Yaskawa INFORM job: A_ROOF_UPPER_0614_2_PAINT_0.JBI

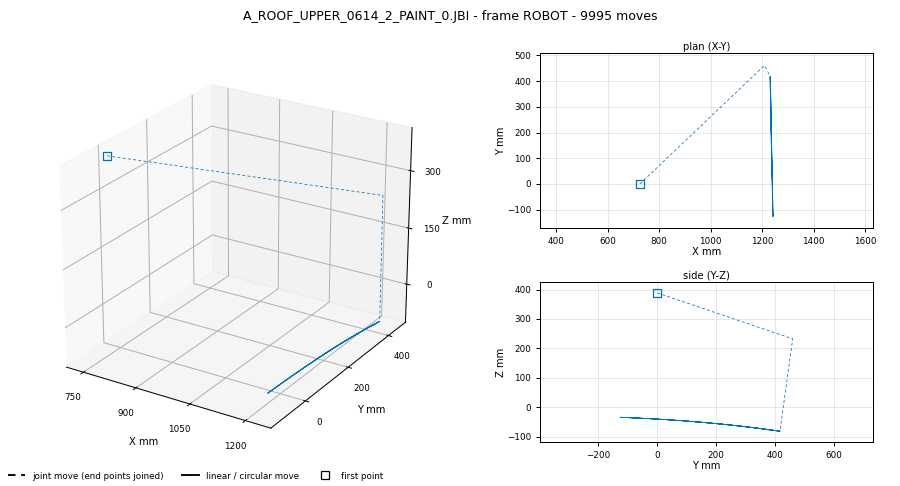
[picture p0: tool path of A_ROOF_UPPER_0614_2_PAINT_0.JBI in frame ROBOT, 9995 of 9995 moves have a stored position in this frame; points joined in program order, loops and branches not executed]
/JOB
//NAME A_ROOF_UPPER_0614_2_PAINT
//POS
///NPOS 9995,0,0,0,0,0
///TOOL 0
///USER 0
///POSTYPE ROBOT
///RECTAN
///RCONF 1,0,0,0,0,0,0,0,0,0,0,0,0,0,0,0,0,0,0,0,0,0,0,0
C00000=725.000,0.000,388.500,-180.000,-0.000,0.000
///TOOL 1
///USER 0
///POSTYPE ROBOT
///RECTAN
C00001=1208.850,460.483,232.516,-175.614,7.825,148.236
C00002=1232.740,417.098,-81.457,-175.614,7.825,148.236
C00003=1232.746,416.739,-81.407,-175.614,7.822,148.236
C00004=1232.752,416.380,-81.357,-175.615,7.819,148.235
C00005=1232.757,416.020,-81.307,-175.616,7.816,148.234
C00006=1232.764,415.662,-81.256,-175.617,7.813,148.234
C00007=1232.767,415.414,-81.222,-175.617,7.811,148.234
C00008=1232.771,415.166,-81.188,-175.619,7.808,148.233
C00009=1232.775,414.918,-81.153,-175.619,7.806,148.233
C00010=1232.779,414.671,-81.119,-175.619,7.804,148.232
C00011=1232.784,414.424,-81.085,-175.620,7.802,148.232
C00012=1232.788,414.176,-81.050,-175.621,7.800,148.232
C00013=1232.792,413.929,-81.016,-175.621,7.798,148.231
C00014=1232.796,413.680,-80.981,-175.621,7.796,148.231
C00015=1232.800,413.433,-80.947,-175.623,7.793,148.230
C00016=1232.804,413.186,-80.913,-175.623,7.791,148.230
C00017=1232.808,412.938,-80.878,-175.624,7.789,148.230
C00018=1232.813,412.690,-80.843,-175.625,7.787,148.229
C00019=1232.816,412.443,-80.809,-175.625,7.785,148.229
C00020=1232.820,412.195,-80.775,-175.626,7.782,148.228
C00021=1232.825,411.948,-80.740,-175.626,7.780,148.228
C00022=1232.828,411.700,-80.706,-175.627,7.778,148.228
C00023=1232.833,411.452,-80.672,-175.628,7.776,148.227
C00024=1232.836,411.205,-80.637,-175.628,7.774,148.227
C00025=1232.841,410.957,-80.603,-175.629,7.772,148.226
C00026=1232.845,410.710,-80.568,-175.630,7.769,148.226
C00027=1232.848,410.462,-80.534,-175.630,7.767,148.226
C00028=1232.853,410.214,-80.500,-175.631,7.765,148.225
C00029=1232.856,409.966,-80.466,-175.631,7.763,148.225
C00030=1232.861,409.719,-80.432,-175.632,7.760,148.224
C00031=1232.866,409.471,-80.397,-175.633,7.758,148.224
C00032=1232.869,409.224,-80.363,-175.634,7.756,148.224
C00033=1232.873,408.976,-80.329,-175.634,7.754,148.223
C00034=1232.877,408.729,-80.295,-175.634,7.752,148.223
C00035=1232.881,408.481,-80.260,-175.635,7.749,148.222
C00036=1232.886,408.233,-80.225,-175.636,7.747,148.222
C00037=1232.890,407.986,-80.191,-175.637,7.745,148.222
C00038=1232.894,407.738,-80.157,-175.637,7.743,148.221
C00039=1232.898,407.491,-80.123,-175.638,7.740,148.221
C00040=1232.902,407.243,-80.089,-175.639,7.738,148.220
C00041=1232.905,406.995,-80.055,-175.639,7.736,148.220
C00042=1232.910,406.748,-80.020,-175.640,7.734,148.220
C00043=1232.914,406.501,-79.986,-175.641,7.731,148.219
C00044=1232.918,406.253,-79.952,-175.641,7.729,148.219
C00045=1232.923,406.005,-79.918,-175.642,7.727,148.218
C00046=1232.927,405.757,-79.884,-175.643,7.724,148.218
C00047=1232.931,405.509,-79.849,-175.644,7.722,148.218
C00048=1232.934,405.262,-79.815,-175.644,7.720,148.217
C00049=1232.939,405.015,-79.781,-175.644,7.718,148.217
C00050=1232.942,404.766,-79.747,-175.646,7.715,148.216
C00051=1232.947,404.519,-79.713,-175.646,7.713,148.216
C00052=1232.951,404.272,-79.679,-175.647,7.711,148.216
C00053=1232.955,404.024,-79.644,-175.648,7.708,148.215
C00054=1232.959,403.777,-79.610,-175.649,7.706,148.215
C00055=1232.964,403.529,-79.576,-175.649,7.704,148.214
C00056=1232.967,403.281,-79.542,-175.650,7.701,148.214
C00057=1232.971,403.033,-79.508,-175.651,7.699,148.214
C00058=1232.975,402.786,-79.474,-175.651,7.697,148.213
C00059=1232.979,402.538,-79.440,-175.652,7.694,148.213
C00060=1232.983,402.290,-79.406,-175.653,7.692,148.212
C00061=1232.988,402.043,-79.371,-175.653,7.690,148.212
C00062=1232.991,401.795,-79.337,-175.654,7.687,148.212
C00063=1232.996,401.547,-79.303,-175.655,7.685,148.211
C00064=1233.000,401.300,-79.270,-175.656,7.683,148.211
C00065=1233.004,401.053,-79.236,-175.657,7.681,148.211
C00066=1233.008,400.804,-79.202,-175.657,7.678,148.210
C00067=1233.012,400.557,-79.168,-175.658,7.676,148.210
C00068=1233.016,400.310,-79.133,-175.659,7.673,148.209
C00069=1233.020,400.061,-79.100,-175.659,7.671,148.209
C00070=1233.024,399.814,-79.065,-175.660,7.669,148.209
C00071=1233.028,399.567,-79.031,-175.661,7.667,148.208
C00072=1233.033,399.319,-78.998,-175.662,7.665,148.208
C00073=1233.036,399.071,-78.963,-175.662,7.662,148.207
C00074=1233.040,398.824,-78.930,-175.663,7.660,148.207
C00075=1233.045,398.576,-78.896,-175.664,7.658,148.206
C00076=1233.049,398.329,-78.862,-175.665,7.655,148.206
C00077=1233.053,398.080,-78.827,-175.666,7.653,148.206
C00078=1233.057,397.833,-78.794,-175.667,7.650,148.205
C00079=1233.061,397.586,-78.760,-175.667,7.648,148.205
C00080=1233.066,397.338,-78.726,-175.668,7.645,148.204
C00081=1233.069,397.090,-78.692,-175.669,7.643,148.204
C00082=1233.074,396.842,-78.658,-175.669,7.641,148.204
C00083=1233.078,396.595,-78.624,-175.670,7.638,148.203
C00084=1233.081,396.348,-78.591,-175.671,7.636,148.203
C00085=1233.086,396.099,-78.556,-175.672,7.633,148.203
C00086=1233.090,395.852,-78.523,-175.673,7.631,148.202
C00087=1233.094,395.604,-78.489,-175.674,7.628,148.202
C00088=1233.098,395.357,-78.455,-175.674,7.626,148.201
C00089=1233.102,395.108,-78.421,-175.675,7.623,148.201
C00090=1233.106,394.861,-78.388,-175.676,7.621,148.201
C00091=1233.111,394.613,-78.354,-175.677,7.619,148.200
C00092=1233.114,394.366,-78.320,-175.678,7.617,148.200
C00093=1233.119,394.118,-78.286,-175.678,7.615,148.199
C00094=1233.122,393.870,-78.252,-175.680,7.612,148.199
C00095=1233.127,393.589,-78.213,-175.681,7.609,148.199
C00096=1233.132,393.307,-78.175,-175.681,7.606,148.198
C00097=1233.136,393.027,-78.137,-175.682,7.604,148.198
C00098=1233.141,392.746,-78.099,-175.683,7.601,148.197
C00099=1233.145,392.498,-78.065,-175.684,7.598,148.197
C00100=1233.150,392.250,-78.031,-175.685,7.596,148.197
C00101=1233.153,392.003,-77.997,-175.686,7.593,148.196
C00102=1233.158,391.755,-77.964,-175.687,7.591,148.196
C00103=1233.162,391.507,-77.931,-175.688,7.589,148.195
C00104=1233.166,391.259,-77.896,-175.689,7.586,148.195
C00105=1233.170,391.011,-77.863,-175.690,7.584,148.195
C00106=1233.174,390.764,-77.829,-175.691,7.581,148.194
C00107=1233.178,390.516,-77.795,-175.691,7.579,148.194
C00108=1233.183,390.268,-77.762,-175.692,7.576,148.193
C00109=1233.186,390.021,-77.728,-175.693,7.574,148.193
C00110=1233.190,389.773,-77.695,-175.694,7.571,148.193
C00111=1233.195,389.525,-77.660,-175.695,7.569,148.192
C00112=1233.199,389.278,-77.627,-175.696,7.566,148.192
C00113=1233.203,389.030,-77.594,-175.697,7.563,148.191
C00114=1233.207,388.783,-77.560,-175.697,7.561,148.191
C00115=1233.212,388.535,-77.526,-175.699,7.559,148.191
C00116=1233.215,388.286,-77.493,-175.699,7.557,148.190
C00117=1233.219,388.039,-77.459,-175.700,7.554,148.190
C00118=1233.223,387.792,-77.426,-175.702,7.551,148.189
C00119=1233.227,387.544,-77.393,-175.702,7.549,148.189
C00120=1233.232,387.296,-77.358,-175.703,7.546,148.189
C00121=1233.236,387.049,-77.325,-175.704,7.544,148.188
C00122=1233.240,386.801,-77.292,-175.705,7.541,148.188
C00123=1233.243,386.553,-77.258,-175.706,7.538,148.188
C00124=1233.247,386.305,-77.224,-175.707,7.536,148.187
C00125=1233.252,386.057,-77.191,-175.708,7.534,148.187
C00126=1233.256,385.810,-77.158,-175.710,7.531,148.187
C00127=1233.260,385.563,-77.124,-175.710,7.529,148.186
C00128=1233.264,385.315,-77.091,-175.711,7.526,148.186
C00129=1233.269,385.067,-77.057,-175.713,7.524,148.186
C00130=1233.273,384.819,-77.024,-175.713,7.522,148.185
C00131=1233.277,384.571,-76.989,-175.714,7.519,148.185
C00132=1233.281,384.324,-76.956,-175.715,7.517,148.184
C00133=1233.285,384.076,-76.923,-175.716,7.514,148.184
C00134=1233.289,383.828,-76.890,-175.717,7.511,148.184
C00135=1233.293,383.580,-76.857,-175.719,7.508,148.183
C00136=1233.297,383.333,-76.823,-175.719,7.506,148.183
C00137=1233.301,383.086,-76.790,-175.720,7.503,148.182
C00138=1233.306,382.837,-76.756,-175.721,7.501,148.182
C00139=1233.310,382.590,-76.723,-175.723,7.499,148.182
C00140=1233.314,382.341,-76.689,-175.724,7.496,148.182
C00141=1233.318,382.094,-76.656,-175.725,7.493,148.181
C00142=1233.322,381.846,-76.623,-175.725,7.491,148.181
C00143=1233.326,381.599,-76.589,-175.727,7.488,148.180
C00144=1233.330,381.351,-76.556,-175.728,7.486,148.180
C00145=1233.334,381.103,-76.523,-175.729,7.483,148.180
C00146=1233.338,380.856,-76.490,-175.730,7.481,148.179
C00147=1233.342,380.608,-76.457,-175.731,7.478,148.179
C00148=1233.347,380.360,-76.423,-175.732,7.475,148.179
C00149=1233.351,380.112,-76.390,-175.733,7.473,148.178
C00150=1233.356,379.864,-76.356,-175.734,7.471,148.178
C00151=1233.360,379.617,-76.323,-175.735,7.468,148.178
C00152=1233.364,379.369,-76.290,-175.736,7.465,148.177
C00153=1233.368,379.121,-76.257,-175.738,7.462,148.177
C00154=1233.372,378.874,-76.223,-175.739,7.460,148.177
C00155=1233.376,378.626,-76.190,-175.740,7.458,148.176
C00156=1233.379,378.378,-76.156,-175.741,7.455,148.176
C00157=1233.384,378.130,-76.123,-175.742,7.452,148.175
C00158=1233.388,377.882,-76.090,-175.743,7.450,148.175
C00159=1233.392,377.635,-76.057,-175.744,7.447,148.175
C00160=1233.396,377.387,-76.024,-175.746,7.445,148.174
C00161=1233.400,377.139,-75.991,-175.747,7.442,148.174
C00162=1233.404,376.891,-75.957,-175.748,7.439,148.174
C00163=1233.408,376.644,-75.924,-175.749,7.437,148.173
C00164=1233.413,376.395,-75.892,-175.750,7.434,148.173
C00165=1233.417,376.148,-75.859,-175.751,7.432,148.173
C00166=1233.421,375.900,-75.826,-175.753,7.429,148.173
C00167=1233.425,375.652,-75.792,-175.754,7.426,148.172
C00168=1233.429,375.404,-75.759,-175.755,7.423,148.172
C00169=1233.434,375.157,-75.726,-175.756,7.421,148.171
C00170=1233.438,374.909,-75.693,-175.757,7.419,148.171
C00171=1233.442,374.661,-75.660,-175.759,7.416,148.171
C00172=1233.446,374.414,-75.627,-175.760,7.413,148.170
C00173=1233.450,374.166,-75.594,-175.761,7.411,148.170
C00174=1233.454,373.918,-75.560,-175.763,7.408,148.170
C00175=1233.458,373.670,-75.528,-175.763,7.406,148.169
C00176=1233.462,373.422,-75.495,-175.765,7.403,148.169
C00177=1233.466,373.175,-75.462,-175.766,7.401,148.169
C00178=1233.470,372.927,-75.429,-175.767,7.398,148.168
C00179=1233.474,372.679,-75.396,-175.769,7.395,148.168
C00180=1233.479,372.431,-75.363,-175.770,7.392,148.168
C00181=1233.483,372.183,-75.330,-175.771,7.390,148.168
C00182=1233.487,371.935,-75.297,-175.773,7.387,148.167
C00183=1233.492,371.688,-75.264,-175.773,7.385,148.167
C00184=1233.496,371.441,-75.231,-175.775,7.383,148.167
C00185=1233.499,371.193,-75.199,-175.776,7.380,148.166
C00186=1233.504,370.945,-75.166,-175.777,7.377,148.166
C00187=1233.508,370.697,-75.133,-175.779,7.374,148.166
C00188=1233.512,370.449,-75.100,-175.780,7.371,148.165
C00189=1233.516,370.202,-75.067,-175.782,7.369,148.165
C00190=1233.521,369.953,-75.034,-175.783,7.366,148.165
C00191=1233.525,369.706,-75.001,-175.784,7.364,148.165
C00192=1233.528,369.458,-74.969,-175.785,7.361,148.164
C00193=1233.532,369.210,-74.935,-175.787,7.358,148.164
C00194=1233.537,368.962,-74.903,-175.788,7.355,148.164
C00195=1233.541,368.714,-74.870,-175.790,7.353,148.163
C00196=1233.545,368.467,-74.837,-175.790,7.351,148.163
C00197=1233.549,368.219,-74.805,-175.792,7.348,148.163
C00198=1233.554,367.972,-74.772,-175.793,7.346,148.162
C00199=1233.558,367.692,-74.734,-175.795,7.342,148.162
C00200=1233.563,367.412,-74.698,-175.797,7.339,148.162
C00201=1233.568,367.133,-74.661,-175.798,7.336,148.161
C00202=1233.572,366.854,-74.624,-175.800,7.333,148.161
C00203=1233.577,366.605,-74.591,-175.801,7.330,148.161
C00204=1233.580,366.358,-74.559,-175.803,7.328,148.161
C00205=1233.585,366.110,-74.526,-175.804,7.325,148.160
C00206=1233.589,365.862,-74.493,-175.805,7.322,148.160
C00207=1233.594,365.614,-74.461,-175.807,7.320,148.160
C00208=1233.597,365.367,-74.428,-175.808,7.317,148.159
C00209=1233.601,365.119,-74.395,-175.810,7.314,148.159
C00210=1233.606,364.871,-74.363,-175.811,7.312,148.159
C00211=1233.610,364.623,-74.330,-175.813,7.309,148.159
C00212=1233.614,364.376,-74.298,-175.814,7.307,148.158
C00213=1233.618,364.128,-74.265,-175.815,7.304,148.158
C00214=1233.623,363.879,-74.233,-175.817,7.301,148.158
C00215=1233.626,363.632,-74.200,-175.818,7.298,148.157
C00216=1233.631,363.384,-74.168,-175.820,7.296,148.157
C00217=1233.635,363.136,-74.134,-175.821,7.293,148.157
C00218=1233.639,362.889,-74.103,-175.823,7.291,148.157
C00219=1233.643,362.641,-74.070,-175.824,7.288,148.156
C00220=1233.648,362.393,-74.037,-175.826,7.285,148.156
C00221=1233.651,362.145,-74.005,-175.827,7.283,148.156
C00222=1233.655,361.897,-73.972,-175.829,7.280,148.156
C00223=1233.660,361.648,-73.940,-175.830,7.278,148.156
C00224=1233.664,361.402,-73.908,-175.831,7.275,148.155
C00225=1233.668,361.153,-73.875,-175.833,7.272,148.155
C00226=1233.672,360.906,-73.842,-175.835,7.270,148.155
C00227=1233.676,360.658,-73.810,-175.836,7.267,148.155
C00228=1233.681,360.409,-73.778,-175.837,7.264,148.154
C00229=1233.685,360.162,-73.745,-175.839,7.262,148.154
C00230=1233.689,359.914,-73.713,-175.841,7.259,148.154
C00231=1233.693,359.666,-73.681,-175.842,7.257,148.154
C00232=1233.697,359.418,-73.648,-175.843,7.254,148.153
C00233=1233.702,359.171,-73.616,-175.846,7.250,148.153
C00234=1233.706,358.922,-73.584,-175.847,7.248,148.153
C00235=1233.710,358.675,-73.551,-175.849,7.245,148.153
C00236=1233.714,358.427,-73.519,-175.850,7.243,148.152
C00237=1233.718,358.179,-73.487,-175.852,7.240,148.152
C00238=1233.723,357.932,-73.454,-175.853,7.238,148.152
C00239=1233.727,357.683,-73.422,-175.855,7.235,148.152
C00240=1233.731,357.435,-73.390,-175.856,7.232,148.151
C00241=1233.735,357.187,-73.357,-175.858,7.230,148.151
C00242=1233.739,356.940,-73.325,-175.859,7.227,148.151
C00243=1233.744,356.692,-73.293,-175.861,7.225,148.151
C00244=1233.747,356.444,-73.261,-175.862,7.222,148.150
C00245=1233.752,356.195,-73.228,-175.865,7.219,148.150
C00246=1233.756,355.949,-73.196,-175.866,7.216,148.150
C00247=1233.760,355.700,-73.164,-175.868,7.214,148.150
C00248=1233.764,355.452,-73.132,-175.869,7.211,148.150
C00249=1233.769,355.205,-73.100,-175.871,7.208,148.149
C00250=1233.773,354.957,-73.068,-175.872,7.206,148.149
C00251=1233.777,354.708,-73.035,-175.874,7.203,148.149
C00252=1233.781,354.461,-73.003,-175.875,7.201,148.149
C00253=1233.786,354.213,-72.971,-175.877,7.198,148.149
C00254=1233.789,353.965,-72.939,-175.879,7.196,148.148
C00255=1233.794,353.717,-72.907,-175.881,7.192,148.148
C00256=1233.798,353.469,-72.875,-175.882,7.190,148.148
C00257=1233.802,353.221,-72.843,-175.884,7.187,148.148
C00258=1233.806,352.973,-72.811,-175.886,7.185,148.148
C00259=1233.810,352.725,-72.779,-175.887,7.182,148.147
C00260=1233.815,352.477,-72.747,-175.889,7.180,148.147
C00261=1233.819,352.229,-72.715,-175.891,7.177,148.147
C00262=1233.823,351.981,-72.683,-175.892,7.174,148.147
C00263=1233.827,351.734,-72.650,-175.894,7.171,148.147
C00264=1233.831,351.486,-72.619,-175.896,7.169,148.146
C00265=1233.835,351.238,-72.586,-175.898,7.166,148.146
C00266=1233.840,350.991,-72.555,-175.899,7.163,148.146
C00267=1233.843,350.743,-72.523,-175.901,7.161,148.146
C00268=1233.848,350.494,-72.490,-175.902,7.158,148.146
C00269=1233.852,350.247,-72.459,-175.904,7.156,148.145
C00270=1233.856,349.999,-72.427,-175.906,7.152,148.145
C00271=1233.861,349.750,-72.395,-175.908,7.150,148.145
C00272=1233.865,349.502,-72.364,-175.909,7.147,148.145
C00273=1233.869,349.254,-72.332,-175.911,7.145,148.145
C00274=1233.874,349.007,-72.300,-175.913,7.142,148.145
C00275=1233.877,348.759,-72.268,-175.914,7.140,148.144
C00276=1233.881,348.511,-72.236,-175.916,7.137,148.144
C00277=1233.886,348.263,-72.204,-175.918,7.134,148.144
C00278=1233.890,348.015,-72.172,-175.920,7.131,148.144
C00279=1233.893,347.767,-72.140,-175.921,7.129,148.144
C00280=1233.898,347.519,-72.108,-175.923,7.127,148.144
C00281=1233.902,347.271,-72.077,-175.925,7.124,148.143
C00282=1233.907,347.023,-72.046,-175.927,7.122,148.143
C00283=1233.911,346.775,-72.014,-175.929,7.118,148.143
C00284=1233.915,346.527,-71.981,-175.930,7.116,148.143
C00285=1233.919,346.280,-71.950,-175.932,7.113,148.143
C00286=1233.923,346.032,-71.918,-175.934,7.111,148.142
C00287=1233.928,345.784,-71.887,-175.936,7.108,148.142
C00288=1233.932,345.535,-71.855,-175.937,7.106,148.142
C00289=1233.936,345.287,-71.823,-175.940,7.102,148.142
C00290=1233.940,345.040,-71.792,-175.941,7.100,148.142
C00291=1233.944,344.792,-71.760,-175.943,7.097,148.142
C00292=1233.948,344.544,-71.729,-175.944,7.095,148.141
C00293=1233.953,344.296,-71.697,-175.947,7.093,148.142
C00294=1233.957,344.048,-71.665,-175.948,7.090,148.141
C00295=1233.961,343.800,-71.634,-175.950,7.087,148.141
C00296=1233.965,343.552,-71.602,-175.952,7.084,148.141
C00297=1233.969,343.304,-71.571,-175.954,7.082,148.141
C00298=1233.974,343.056,-71.538,-175.956,7.079,148.141
C00299=1233.978,342.808,-71.507,-175.957,7.077,148.141
C00300=1233.982,342.560,-71.476,-175.959,7.073,148.140
C00301=1233.986,342.313,-71.444,-175.961,7.071,148.140
C00302=1233.990,342.064,-71.413,-175.963,7.069,148.140
C00303=1233.995,341.787,-71.378,-175.965,7.066,148.140
C00304=1234.000,341.509,-71.343,-175.967,7.063,148.140
C00305=1234.004,341.231,-71.307,-175.970,7.060,148.140
C00306=1234.009,340.955,-71.272,-175.971,7.057,148.140
C00307=1234.013,340.706,-71.241,-175.973,7.055,148.139
C00308=1234.018,340.458,-71.209,-175.975,7.052,148.139
C00309=1234.022,340.210,-71.178,-175.977,7.049,148.139
C00310=1234.026,339.962,-71.146,-175.979,7.047,148.139
C00311=1234.030,339.714,-71.115,-175.980,7.044,148.139
C00312=1234.035,339.466,-71.084,-175.982,7.042,148.139
C00313=1234.038,339.218,-71.052,-175.985,7.038,148.139
C00314=1234.043,338.970,-71.021,-175.986,7.036,148.138
C00315=1234.047,338.722,-70.989,-175.988,7.034,148.139
C00316=1234.051,338.474,-70.958,-175.990,7.031,148.138
C00317=1234.056,338.227,-70.927,-175.992,7.029,148.138
C00318=1234.060,337.978,-70.896,-175.994,7.025,148.138
C00319=1234.064,337.730,-70.865,-175.996,7.023,148.138
C00320=1234.068,337.482,-70.833,-175.998,7.021,148.138
C00321=1234.073,337.234,-70.802,-175.999,7.018,148.138
C00322=1234.076,336.986,-70.771,-176.001,7.016,148.138
C00323=1234.081,336.738,-70.740,-176.004,7.013,148.138
C00324=1234.085,336.490,-70.708,-176.005,7.010,148.137
C00325=1234.089,336.242,-70.677,-176.007,7.008,148.137
C00326=1234.094,335.994,-70.646,-176.009,7.005,148.137
C00327=1234.098,335.746,-70.615,-176.011,7.003,148.137
C00328=1234.102,335.498,-70.584,-176.013,7.000,148.137
C00329=1234.106,335.250,-70.553,-176.015,6.997,148.137
C00330=1234.110,335.002,-70.521,-176.017,6.995,148.137
C00331=1234.114,334.754,-70.490,-176.019,6.992,148.137
C00332=1234.119,334.506,-70.459,-176.021,6.989,148.137
C00333=1234.123,334.258,-70.428,-176.023,6.987,148.137
C00334=1234.127,334.010,-70.397,-176.025,6.985,148.137
C00335=1234.132,333.762,-70.366,-176.027,6.982,148.136
C00336=1234.136,333.514,-70.334,-176.029,6.980,148.136
C00337=1234.140,333.266,-70.303,-176.031,6.976,148.136
C00338=1234.145,333.018,-70.273,-176.033,6.974,148.136
C00339=1234.148,332.769,-70.242,-176.035,6.972,148.136
C00340=1234.153,332.522,-70.211,-176.037,6.969,148.136
C00341=1234.157,332.274,-70.180,-176.038,6.967,148.136
C00342=1234.161,332.025,-70.149,-176.041,6.964,148.136
C00343=1234.166,331.778,-70.118,-176.043,6.961,148.136
C00344=1234.170,331.530,-70.087,-176.045,6.959,148.136
C00345=1234.174,331.282,-70.055,-176.046,6.956,148.136
C00346=1234.178,331.034,-70.025,-176.049,6.953,148.136
C00347=1234.183,330.786,-69.994,-176.050,6.951,148.135
C00348=1234.187,330.537,-69.963,-176.053,6.949,148.135
C00349=1234.191,330.289,-69.932,-176.054,6.946,148.135
C00350=1234.196,330.041,-69.902,-176.056,6.944,148.135
C00351=1234.200,329.793,-69.870,-176.059,6.941,148.135
C00352=1234.203,329.546,-69.840,-176.061,6.938,148.135
C00353=1234.208,329.298,-69.809,-176.063,6.936,148.135
C00354=1234.212,329.049,-69.778,-176.064,6.933,148.135
C00355=1234.217,328.801,-69.747,-176.067,6.930,148.135
C00356=1234.221,328.553,-69.716,-176.069,6.928,148.135
C00357=1234.225,328.305,-69.686,-176.071,6.926,148.135
C00358=1234.229,328.057,-69.655,-176.073,6.923,148.135
C00359=1234.234,327.809,-69.624,-176.075,6.920,148.135
C00360=1234.238,327.560,-69.593,-176.077,6.918,148.135
C00361=1234.242,327.313,-69.563,-176.079,6.916,148.135
C00362=1234.246,327.065,-69.532,-176.081,6.913,148.135
C00363=1234.251,326.817,-69.501,-176.083,6.911,148.135
C00364=1234.254,326.568,-69.471,-176.085,6.907,148.134
C00365=1234.259,326.320,-69.440,-176.087,6.905,148.134
C00366=1234.263,326.072,-69.409,-176.089,6.903,148.134
C00367=1234.268,325.824,-69.379,-176.091,6.900,148.134
C00368=1234.271,325.576,-69.348,-176.093,6.897,148.134
C00369=1234.276,325.328,-69.317,-176.095,6.895,148.134
C00370=1234.280,325.080,-69.286,-176.098,6.893,148.134
C00371=1234.284,324.833,-69.256,-176.099,6.890,148.134
C00372=1234.289,324.583,-69.226,-176.101,6.888,148.134
C00373=1234.293,324.335,-69.195,-176.104,6.885,148.134
C00374=1234.297,324.088,-69.165,-176.106,6.883,148.134
C00375=1234.302,323.840,-69.134,-176.108,6.880,148.134
C00376=1234.306,323.591,-69.103,-176.110,6.878,148.134
C00377=1234.310,323.343,-69.073,-176.112,6.875,148.134
C00378=1234.314,323.095,-69.042,-176.114,6.872,148.134
C00379=1234.319,322.847,-69.012,-176.116,6.870,148.134
C00380=1234.323,322.599,-68.982,-176.118,6.868,148.134
C00381=1234.327,322.351,-68.951,-176.120,6.865,148.134
C00382=1234.331,322.103,-68.921,-176.122,6.862,148.134
C00383=1234.336,321.855,-68.890,-176.125,6.860,148.134
C00384=1234.341,321.606,-68.860,-176.127,6.858,148.134
C00385=1234.344,321.359,-68.830,-176.128,6.855,148.134
C00386=1234.349,321.111,-68.799,-176.131,6.852,148.134
C00387=1234.353,320.862,-68.769,-176.133,6.850,148.134
C00388=1234.357,320.614,-68.738,-176.135,6.848,148.134
C00389=1234.361,320.366,-68.708,-176.137,6.846,148.134
C00390=1234.366,320.118,-68.677,-176.139,6.842,148.134
C00391=1234.370,319.870,-68.648,-176.141,6.840,148.134
C00392=1234.374,319.622,-68.617,-176.144,6.838,148.134
C00393=1234.378,319.373,-68.586,-176.146,6.836,148.134
C00394=1234.383,319.125,-68.557,-176.148,6.833,148.134
C00395=1234.387,318.877,-68.526,-176.150,6.830,148.134
C00396=1234.391,318.629,-68.496,-176.152,6.828,148.134
C00397=1234.396,318.381,-68.466,-176.154,6.826,148.134
C00398=1234.400,318.133,-68.435,-176.156,6.823,148.134
C00399=1234.405,317.885,-68.405,-176.159,6.820,148.134
C00400=1234.409,317.637,-68.375,-176.161,6.818,148.134
C00401=1234.412,317.388,-68.345,-176.163,6.815,148.134
C00402=1234.417,317.140,-68.315,-176.165,6.813,148.134
C00403=1234.421,316.892,-68.284,-176.167,6.810,148.134
C00404=1234.426,316.644,-68.254,-176.169,6.808,148.134
C00405=1234.430,316.396,-68.224,-176.171,6.806,148.134
C00406=1234.435,316.148,-68.194,-176.174,6.803,148.134
C00407=1234.439,315.872,-68.160,-176.176,6.800,148.134
C00408=1234.444,315.596,-68.127,-176.178,6.798,148.134
C00409=1234.448,315.321,-68.094,-176.181,6.795,148.134
C00410=1234.453,315.046,-68.061,-176.184,6.792,148.134
C00411=1234.458,314.796,-68.031,-176.186,6.790,148.134
C00412=1234.461,314.549,-68.000,-176.188,6.788,148.134
C00413=1234.466,314.300,-67.970,-176.189,6.785,148.134
C00414=1234.470,314.052,-67.940,-176.192,6.782,148.134
C00415=1234.474,313.804,-67.911,-176.194,6.780,148.134
C00416=1234.479,313.556,-67.880,-176.196,6.778,148.134
C00417=1234.483,313.308,-67.851,-176.198,6.775,148.134
C00418=1234.487,313.060,-67.821,-176.200,6.773,148.134
C00419=1234.492,312.812,-67.790,-176.203,6.770,148.134
C00420=1234.496,312.563,-67.761,-176.205,6.768,148.134
C00421=1234.500,312.315,-67.731,-176.207,6.766,148.134
C00422=1234.504,312.068,-67.701,-176.209,6.763,148.134
C00423=1234.509,311.819,-67.671,-176.212,6.760,148.134
C00424=1234.513,311.571,-67.642,-176.214,6.758,148.134
C00425=1234.517,311.323,-67.612,-176.216,6.756,148.134
C00426=1234.522,311.074,-67.581,-176.218,6.754,148.134
C00427=1234.526,310.826,-67.552,-176.220,6.751,148.134
C00428=1234.530,310.579,-67.522,-176.223,6.748,148.134
C00429=1234.534,310.330,-67.492,-176.225,6.746,148.134
C00430=1234.539,310.082,-67.462,-176.227,6.744,148.134
C00431=1234.543,309.833,-67.433,-176.229,6.742,148.134
C00432=1234.547,309.586,-67.403,-176.232,6.739,148.134
C00433=1234.552,309.338,-67.373,-176.234,6.736,148.135
C00434=1234.556,309.089,-67.344,-176.236,6.734,148.135
C00435=1234.561,308.841,-67.314,-176.238,6.732,148.135
C00436=1234.565,308.592,-67.284,-176.240,6.730,148.135
C00437=1234.569,308.345,-67.254,-176.243,6.727,148.135
C00438=1234.573,308.096,-67.225,-176.245,6.724,148.135
C00439=1234.577,307.848,-67.195,-176.247,6.722,148.135
C00440=1234.582,307.600,-67.165,-176.249,6.720,148.135
C00441=1234.586,307.351,-67.136,-176.251,6.718,148.135
C00442=1234.590,307.103,-67.106,-176.254,6.715,148.135
C00443=1234.595,306.855,-67.077,-176.256,6.712,148.135
C00444=1234.598,306.607,-67.047,-176.258,6.710,148.135
C00445=1234.603,306.359,-67.017,-176.260,6.708,148.135
C00446=1234.607,306.111,-66.988,-176.262,6.706,148.135
C00447=1234.612,305.862,-66.958,-176.266,6.703,148.135
C00448=1234.616,305.615,-66.929,-176.268,6.701,148.135
C00449=1234.621,305.366,-66.899,-176.270,6.698,148.135
C00450=1234.625,305.118,-66.870,-176.272,6.696,148.135
C00451=1234.629,304.870,-66.840,-176.274,6.694,148.136
C00452=1234.633,304.621,-66.811,-176.277,6.691,148.136
C00453=1234.637,304.373,-66.781,-176.279,6.689,148.136
C00454=1234.642,304.125,-66.752,-176.281,6.686,148.136
C00455=1234.646,303.877,-66.722,-176.283,6.684,148.136
C00456=1234.650,303.628,-66.693,-176.286,6.681,148.136
C00457=1234.654,303.380,-66.664,-176.288,6.679,148.136
C00458=1234.659,303.133,-66.634,-176.290,6.677,148.136
C00459=1234.664,302.884,-66.604,-176.292,6.675,148.136
C00460=1234.668,302.636,-66.575,-176.294,6.673,148.136
C00461=1234.672,302.387,-66.546,-176.297,6.670,148.136
C00462=1234.677,302.139,-66.517,-176.299,6.667,148.136
C00463=1234.681,301.890,-66.487,-176.301,6.665,148.136
C00464=1234.685,301.642,-66.458,-176.304,6.663,148.137
C00465=1234.690,301.394,-66.429,-176.306,6.661,148.137
C00466=1234.694,301.146,-66.399,-176.308,6.659,148.137
C00467=1234.698,300.898,-66.370,-176.311,6.656,148.137
C00468=1234.703,300.649,-66.341,-176.313,6.653,148.137
C00469=1234.707,300.401,-66.312,-176.315,6.651,148.137
C00470=1234.710,300.153,-66.283,-176.318,6.649,148.137
C00471=1234.715,299.905,-66.254,-176.320,6.647,148.137
C00472=1234.719,299.657,-66.224,-176.322,6.644,148.137
C00473=1234.724,299.408,-66.196,-176.324,6.642,148.137
C00474=1234.728,299.160,-66.166,-176.326,6.640,148.137
C00475=1234.732,298.912,-66.137,-176.329,6.638,148.137
C00476=1234.737,298.664,-66.108,-176.331,6.635,148.138
C00477=1234.741,298.415,-66.079,-176.334,6.632,148.138
C00478=1234.746,298.167,-66.049,-176.336,6.630,148.138
C00479=1234.750,297.919,-66.020,-176.338,6.628,148.138
C00480=1234.754,297.670,-65.990,-176.341,6.626,148.138
C00481=1234.759,297.422,-65.962,-176.343,6.624,148.138
C00482=1234.762,297.174,-65.933,-176.345,6.622,148.138
C00483=1234.767,296.926,-65.904,-176.347,6.618,148.138
C00484=1234.771,296.677,-65.875,-176.350,6.617,148.138
C00485=1234.776,296.429,-65.846,-176.352,6.614,148.138
C00486=1234.780,296.181,-65.817,-176.354,6.612,148.138
C00487=1234.785,295.932,-65.788,-176.356,6.610,148.138
C00488=1234.789,295.684,-65.758,-176.359,6.607,148.139
C00489=1234.793,295.436,-65.731,-176.362,6.605,148.139
C00490=1234.797,295.188,-65.701,-176.364,6.603,148.139
C00491=1234.802,294.939,-65.672,-176.366,6.600,148.139
C00492=1234.807,294.691,-65.643,-176.368,6.599,148.139
C00493=1234.811,294.443,-65.614,-176.370,6.596,148.139
C00494=1234.814,294.195,-65.586,-176.373,6.593,148.139
C00495=1234.819,293.946,-65.556,-176.376,6.591,148.140
C00496=1234.824,293.698,-65.528,-176.378,6.589,148.140
C00497=1234.828,293.450,-65.498,-176.380,6.587,148.140
C00498=1234.832,293.201,-65.470,-176.382,6.585,148.140
C00499=1234.836,292.954,-65.441,-176.385,6.583,148.140
C00500=1234.841,292.705,-65.412,-176.387,6.580,148.140
C00501=1234.845,292.457,-65.383,-176.389,6.577,148.140
C00502=1234.849,292.209,-65.355,-176.392,6.576,148.140
C00503=1234.854,291.960,-65.326,-176.394,6.573,148.140
C00504=1234.858,291.712,-65.297,-176.396,6.571,148.140
C00505=1234.863,291.463,-65.269,-176.399,6.569,148.141
C00506=1234.867,291.215,-65.240,-176.401,6.567,148.141
C00507=1234.871,290.966,-65.211,-176.403,6.564,148.141
C00508=1234.876,290.718,-65.183,-176.406,6.562,148.141
C00509=1234.880,290.470,-65.154,-176.408,6.560,148.141
C00510=1234.884,290.221,-65.125,-176.410,6.558,148.141
C00511=1234.889,289.947,-65.093,-176.413,6.555,148.141
C00512=1234.894,289.674,-65.061,-176.416,6.553,148.142
C00513=1234.899,289.400,-65.030,-176.418,6.551,148.142
C00514=1234.903,289.126,-64.999,-176.421,6.548,148.142
C00515=1234.908,288.877,-64.970,-176.423,6.546,148.142
C00516=1234.912,288.629,-64.941,-176.425,6.543,148.142
C00517=1234.916,288.381,-64.913,-176.428,6.541,148.142
C00518=1234.921,288.132,-64.884,-176.431,6.538,148.142
C00519=1234.926,287.884,-64.856,-176.433,6.536,148.142
C00520=1234.930,287.636,-64.827,-176.435,6.534,148.143
C00521=1234.934,287.387,-64.798,-176.437,6.532,148.143
C00522=1234.938,287.139,-64.770,-176.440,6.530,148.143
C00523=1234.943,286.891,-64.742,-176.442,6.528,148.143
C00524=1234.947,286.642,-64.714,-176.444,6.526,148.143
C00525=1234.951,286.395,-64.685,-176.446,6.524,148.143
C00526=1234.956,286.146,-64.656,-176.450,6.521,148.144
C00527=1234.960,285.897,-64.628,-176.452,6.519,148.144
C00528=1234.965,285.649,-64.599,-176.454,6.517,148.144
C00529=1234.969,285.400,-64.571,-176.456,6.514,148.144
C00530=1234.974,285.152,-64.543,-176.459,6.513,148.144
C00531=1234.977,284.904,-64.514,-176.461,6.510,148.144
C00532=1234.982,284.656,-64.486,-176.463,6.508,148.144
C00533=1234.986,284.407,-64.458,-176.466,6.505,148.145
C00534=1234.991,284.159,-64.429,-176.468,6.503,148.145
C00535=1234.995,283.911,-64.401,-176.471,6.501,148.145
C00536=1235.000,283.662,-64.373,-176.473,6.499,148.145
C00537=1235.004,283.414,-64.345,-176.476,6.497,148.145
C00538=1235.008,283.165,-64.316,-176.478,6.495,148.145
C00539=1235.012,282.917,-64.288,-176.480,6.493,148.145
C00540=1235.016,282.669,-64.260,-176.482,6.491,148.146
C00541=1235.021,282.420,-64.231,-176.485,6.489,148.146
C00542=1235.025,282.172,-64.203,-176.488,6.486,148.146
C00543=1235.030,281.924,-64.175,-176.490,6.484,148.146
C00544=1235.034,281.675,-64.147,-176.492,6.482,148.146
C00545=1235.039,281.427,-64.118,-176.494,6.479,148.146
C00546=1235.043,281.178,-64.090,-176.497,6.477,148.147
C00547=1235.047,280.930,-64.063,-176.499,6.475,148.147
C00548=1235.052,280.681,-64.034,-176.502,6.473,148.147
C00549=1235.056,280.434,-64.006,-176.504,6.471,148.147
C00550=1235.061,280.185,-63.978,-176.506,6.469,148.147
C00551=1235.065,279.937,-63.950,-176.509,6.466,148.147
C00552=1235.069,279.689,-63.922,-176.512,6.464,148.148
C00553=1235.074,279.439,-63.894,-176.514,6.462,148.148
C00554=1235.078,279.192,-63.866,-176.516,6.460,148.148
C00555=1235.082,278.943,-63.838,-176.519,6.458,148.148
C00556=1235.087,278.695,-63.809,-176.521,6.456,148.148
C00557=1235.091,278.446,-63.781,-176.523,6.454,148.149
C00558=1235.095,278.198,-63.753,-176.526,6.452,148.149
C00559=1235.101,277.950,-63.726,-176.528,6.450,148.149
C00560=1235.104,277.701,-63.698,-176.531,6.448,148.149
C00561=1235.109,277.453,-63.670,-176.533,6.446,148.149
C00562=1235.113,277.204,-63.641,-176.536,6.443,148.149
C00563=1235.117,276.956,-63.613,-176.538,6.441,148.150
C00564=1235.122,276.707,-63.586,-176.540,6.439,148.150
C00565=1235.126,276.459,-63.558,-176.543,6.436,148.150
C00566=1235.131,276.211,-63.530,-176.545,6.435,148.150
C00567=1235.135,275.962,-63.502,-176.547,6.432,148.150
C00568=1235.139,275.714,-63.475,-176.550,6.430,148.151
C00569=1235.143,275.465,-63.446,-176.552,6.428,148.151
C00570=1235.148,275.217,-63.418,-176.555,6.426,148.151
C00571=1235.153,274.969,-63.391,-176.557,6.424,148.151
C00572=1235.157,274.720,-63.363,-176.559,6.422,148.151
C00573=1235.161,274.472,-63.335,-176.562,6.420,148.152
C00574=1235.166,274.223,-63.307,-176.565,6.417,148.152
C00575=1235.170,273.975,-63.279,-176.567,6.415,148.152
C00576=1235.174,273.727,-63.252,-176.569,6.413,148.152
C00577=1235.179,273.479,-63.224,-176.572,6.411,148.152
C00578=1235.183,273.230,-63.196,-176.574,6.409,148.152
C00579=1235.188,272.981,-63.169,-176.577,6.407,148.153
C00580=1235.193,272.733,-63.141,-176.579,6.405,148.153
C00581=1235.196,272.485,-63.113,-176.581,6.403,148.153
C00582=1235.201,272.236,-63.086,-176.584,6.401,148.153
C00583=1235.205,271.988,-63.058,-176.586,6.399,148.153
C00584=1235.209,271.739,-63.031,-176.589,6.397,148.154
C00585=1235.214,271.491,-63.003,-176.591,6.395,148.154
C00586=1235.218,271.243,-62.976,-176.593,6.393,148.154
C00587=1235.223,270.994,-62.947,-176.596,6.391,148.154
C00588=1235.228,270.745,-62.920,-176.598,6.389,148.154
C00589=1235.232,270.498,-62.892,-176.601,6.387,148.155
C00590=1235.236,270.248,-62.865,-176.603,6.385,148.155
C00591=1235.240,270.000,-62.837,-176.606,6.382,148.155
C00592=1235.245,269.752,-62.810,-176.608,6.380,148.155
C00593=1235.249,269.503,-62.782,-176.611,6.378,148.155
C00594=1235.253,269.255,-62.755,-176.613,6.376,148.156
C00595=1235.258,269.006,-62.728,-176.616,6.374,148.156
C00596=1235.262,268.758,-62.700,-176.618,6.372,148.156
C00597=1235.266,268.509,-62.672,-176.620,6.370,148.156
C00598=1235.271,268.261,-62.645,-176.623,6.368,148.157
C00599=1235.275,268.013,-62.618,-176.625,6.366,148.157
C00600=1235.280,267.764,-62.590,-176.628,6.364,148.157
C00601=1235.284,267.516,-62.562,-176.630,6.362,148.157
C00602=1235.289,267.267,-62.535,-176.632,6.360,148.157
C00603=1235.293,267.019,-62.508,-176.635,6.358,148.158
C00604=1235.298,266.771,-62.480,-176.637,6.356,148.158
C00605=1235.302,266.522,-62.453,-176.640,6.354,148.158
C00606=1235.306,266.273,-62.426,-176.642,6.352,148.158
C00607=1235.311,266.025,-62.399,-176.644,6.350,148.158
C00608=1235.315,265.777,-62.371,-176.647,6.348,148.159
C00609=1235.320,265.528,-62.344,-176.650,6.346,148.159
C00610=1235.324,265.279,-62.317,-176.652,6.343,148.159
C00611=1235.329,265.031,-62.290,-176.654,6.342,148.159
C00612=1235.333,264.783,-62.262,-176.657,6.340,148.160
C00613=1235.338,264.534,-62.235,-176.659,6.337,148.160
C00614=1235.342,264.286,-62.208,-176.662,6.336,148.160
C00615=1235.346,264.013,-62.178,-176.665,6.333,148.160
C00616=1235.351,263.740,-62.147,-176.667,6.331,148.161
C00617=1235.356,263.468,-62.118,-176.670,6.329,148.161
C00618=1235.361,263.195,-62.089,-176.672,6.327,148.161
C00619=1235.365,262.946,-62.061,-176.675,6.325,148.161
C00620=1235.370,262.699,-62.034,-176.677,6.323,148.162
C00621=1235.374,262.450,-62.007,-176.679,6.321,148.162
C00622=1235.379,262.202,-61.980,-176.683,6.318,148.162
C00623=1235.384,261.953,-61.953,-176.685,6.316,148.162
C00624=1235.387,261.704,-61.926,-176.688,6.314,148.162
C00625=1235.392,261.456,-61.899,-176.690,6.312,148.163
C00626=1235.396,261.207,-61.872,-176.693,6.310,148.163
C00627=1235.401,260.959,-61.844,-176.695,6.308,148.163
C00628=1235.406,260.710,-61.817,-176.697,6.306,148.163
C00629=1235.410,260.462,-61.790,-176.699,6.305,148.164
C00630=1235.414,260.214,-61.764,-176.702,6.303,148.164
C00631=1235.418,259.964,-61.736,-176.704,6.301,148.164
C00632=1235.423,259.716,-61.709,-176.707,6.299,148.164
C00633=1235.428,259.467,-61.682,-176.709,6.297,148.165
C00634=1235.432,259.219,-61.656,-176.712,6.295,148.165
C00635=1235.436,258.971,-61.629,-176.714,6.293,148.165
C00636=1235.441,258.722,-61.602,-176.717,6.291,148.165
C00637=1235.446,258.474,-61.575,-176.719,6.289,148.166
C00638=1235.450,258.226,-61.548,-176.722,6.287,148.166
C00639=1235.454,257.977,-61.521,-176.724,6.285,148.166
C00640=1235.459,257.729,-61.494,-176.726,6.283,148.166
C00641=1235.463,257.480,-61.467,-176.729,6.281,148.167
C00642=1235.467,257.232,-61.441,-176.732,6.279,148.167
C00643=1235.471,256.983,-61.413,-176.734,6.277,148.167
C00644=1235.476,256.734,-61.386,-176.736,6.275,148.167
C00645=1235.480,256.485,-61.360,-176.739,6.273,148.168
C00646=1235.485,256.237,-61.333,-176.742,6.271,148.168
C00647=1235.490,255.988,-61.306,-176.744,6.269,148.168
C00648=1235.494,255.740,-61.280,-176.746,6.267,148.168
C00649=1235.498,255.492,-61.253,-176.749,6.265,148.169
C00650=1235.503,255.243,-61.226,-176.752,6.264,148.169
C00651=1235.507,254.994,-61.200,-176.754,6.261,148.169
C00652=1235.512,254.746,-61.173,-176.756,6.259,148.169
C00653=1235.516,254.497,-61.146,-176.759,6.258,148.170
C00654=1235.520,254.249,-61.119,-176.761,6.256,148.170
C00655=1235.525,254.001,-61.092,-176.764,6.254,148.170
C00656=1235.530,253.752,-61.066,-176.766,6.252,148.170
C00657=1235.534,253.503,-61.039,-176.769,6.250,148.170
C00658=1235.539,253.255,-61.012,-176.771,6.248,148.171
C00659=1235.543,253.006,-60.987,-176.774,6.246,148.171
C00660=1235.547,252.758,-60.960,-176.776,6.244,148.171
C00661=1235.552,252.509,-60.932,-176.779,6.242,148.171
C00662=1235.556,252.261,-60.906,-176.781,6.240,148.172
C00663=1235.561,252.012,-60.880,-176.783,6.239,148.172
C00664=1235.565,251.764,-60.853,-176.786,6.237,148.172
C00665=1235.570,251.515,-60.827,-176.788,6.235,148.173
C00666=1235.574,251.266,-60.800,-176.791,6.233,148.173
C00667=1235.578,251.018,-60.773,-176.793,6.231,148.173
C00668=1235.583,250.769,-60.748,-176.796,6.229,148.173
C00669=1235.587,250.521,-60.721,-176.799,6.227,148.174
C00670=1235.591,250.272,-60.694,-176.801,6.225,148.174
C00671=1235.596,250.023,-60.668,-176.803,6.223,148.174
C00672=1235.601,249.776,-60.642,-176.806,6.221,148.174
C00673=1235.606,249.527,-60.615,-176.808,6.219,148.175
C00674=1235.610,249.278,-60.589,-176.811,6.217,148.175
C00675=1235.615,249.029,-60.562,-176.814,6.216,148.175
C00676=1235.618,248.781,-60.536,-176.816,6.213,148.175
C00677=1235.623,248.532,-60.510,-176.818,6.211,148.176
C00678=1235.627,248.284,-60.483,-176.821,6.210,148.176
C00679=1235.632,248.035,-60.457,-176.823,6.208,148.176
C00680=1235.636,247.787,-60.430,-176.826,6.207,148.177
C00681=1235.641,247.537,-60.404,-176.828,6.204,148.177
C00682=1235.645,247.289,-60.378,-176.830,6.202,148.177
C00683=1235.650,247.041,-60.352,-176.833,6.201,148.177
C00684=1235.655,246.793,-60.325,-176.836,6.199,148.178
C00685=1235.659,246.544,-60.299,-176.838,6.197,148.178
C00686=1235.663,246.295,-60.272,-176.841,6.195,148.178
C00687=1235.668,246.047,-60.247,-176.843,6.193,148.179
C00688=1235.672,245.798,-60.221,-176.846,6.191,148.179
C00689=1235.677,245.549,-60.194,-176.848,6.189,148.179
C00690=1235.681,245.300,-60.168,-176.851,6.187,148.179
C00691=1235.685,245.053,-60.142,-176.853,6.186,148.180
C00692=1235.690,244.804,-60.116,-176.855,6.184,148.180
C00693=1235.694,244.555,-60.090,-176.858,6.182,148.180
C00694=1235.698,244.307,-60.063,-176.861,6.180,148.181
C00695=1235.703,244.058,-60.037,-176.863,6.178,148.181
C00696=1235.708,243.809,-60.011,-176.865,6.176,148.181
C00697=1235.712,243.561,-59.986,-176.868,6.174,148.181
C00698=1235.717,243.312,-59.959,-176.871,6.172,148.182
C00699=1235.721,243.064,-59.933,-176.873,6.171,148.182
C00700=1235.726,242.815,-59.907,-176.876,6.169,148.182
C00701=1235.730,242.566,-59.880,-176.878,6.168,148.183
C00702=1235.734,242.317,-59.854,-176.880,6.166,148.183
C00703=1235.739,242.069,-59.829,-176.883,6.164,148.183
C00704=1235.743,241.821,-59.803,-176.885,6.162,148.183
C00705=1235.748,241.572,-59.776,-176.888,6.160,148.184
C00706=1235.752,241.323,-59.750,-176.890,6.158,148.184
C00707=1235.757,241.075,-59.725,-176.893,6.156,148.184
C00708=1235.762,240.826,-59.699,-176.896,6.154,148.185
C00709=1235.766,240.577,-59.673,-176.898,6.152,148.185
C00710=1235.771,240.328,-59.647,-176.901,6.150,148.185
C00711=1235.775,240.080,-59.621,-176.903,6.149,148.186
C00712=1235.779,239.832,-59.595,-176.905,6.147,148.186
C00713=1235.784,239.583,-59.569,-176.908,6.145,148.186
C00714=1235.789,239.334,-59.543,-176.910,6.143,148.186
C00715=1235.793,239.085,-59.518,-176.913,6.141,148.187
C00716=1235.798,238.837,-59.492,-176.916,6.140,148.187
C00717=1235.802,238.588,-59.466,-176.918,6.138,148.187
C00718=1235.807,238.339,-59.440,-176.921,6.136,148.188
C00719=1235.812,238.069,-59.412,-176.923,6.134,148.188
C00720=1235.816,237.797,-59.384,-176.926,6.132,148.188
C00721=1235.822,237.526,-59.356,-176.929,6.130,148.189
C00722=1235.826,237.254,-59.327,-176.931,6.128,148.189
C00723=1235.830,237.006,-59.301,-176.934,6.126,148.189
C00724=1235.835,236.758,-59.276,-176.936,6.124,148.189
C00725=1235.839,236.509,-59.250,-176.939,6.123,148.190
C00726=1235.844,236.260,-59.225,-176.942,6.121,148.190
C00727=1235.848,236.011,-59.199,-176.944,6.120,148.190
C00728=1235.853,235.763,-59.173,-176.946,6.118,148.191
C00729=1235.857,235.514,-59.148,-176.949,6.116,148.191
C00730=1235.862,235.264,-59.122,-176.952,6.114,148.191
C00731=1235.867,235.016,-59.097,-176.954,6.112,148.192
C00732=1235.871,234.768,-59.071,-176.957,6.110,148.192
C00733=1235.875,234.519,-59.045,-176.959,6.108,148.192
C00734=1235.880,234.271,-59.020,-176.961,6.107,148.193
C00735=1235.884,234.022,-58.994,-176.964,6.105,148.193
C00736=1235.889,233.773,-58.968,-176.966,6.103,148.193
C00737=1235.894,233.525,-58.943,-176.969,6.101,148.193
C00738=1235.898,233.276,-58.917,-176.971,6.099,148.194
C00739=1235.902,233.027,-58.891,-176.974,6.098,148.194
C00740=1235.907,232.779,-58.867,-176.977,6.096,148.194
C00741=1235.911,232.530,-58.841,-176.979,6.095,148.195
C00742=1235.916,232.282,-58.816,-176.981,6.093,148.195
C00743=1235.920,232.033,-58.790,-176.984,6.091,148.195
C00744=1235.925,231.784,-58.764,-176.987,6.089,148.196
C00745=1235.930,231.535,-58.739,-176.989,6.087,148.196
C00746=1235.934,231.287,-58.714,-176.992,6.085,148.196
C00747=1235.938,231.038,-58.688,-176.994,6.084,148.197
C00748=1235.943,230.790,-58.663,-176.996,6.082,148.197
C00749=1235.948,230.540,-58.638,-176.999,6.080,148.197
C00750=1235.952,230.292,-58.612,-177.002,6.078,148.198
C00751=1235.957,230.043,-58.586,-177.004,6.077,148.198
C00752=1235.961,229.794,-58.561,-177.007,6.075,148.198
C00753=1235.965,229.546,-58.537,-177.009,6.074,148.199
C00754=1235.969,229.297,-58.511,-177.012,6.072,148.199
C00755=1235.974,229.049,-58.485,-177.014,6.070,148.199
C00756=1235.979,228.800,-58.460,-177.017,6.068,148.200
C00757=1235.984,228.552,-58.435,-177.019,6.066,148.200
C00758=1235.988,228.303,-58.409,-177.022,6.064,148.200
C00759=1235.992,228.053,-58.384,-177.024,6.063,148.201
C00760=1235.997,227.805,-58.359,-177.027,6.061,148.201
C00761=1236.001,227.557,-58.333,-177.029,6.059,148.201
C00762=1236.006,227.308,-58.309,-177.032,6.058,148.202
C00763=1236.010,227.059,-58.283,-177.035,6.056,148.202
C00764=1236.015,226.811,-58.259,-177.037,6.054,148.202
C00765=1236.019,226.562,-58.233,-177.039,6.053,148.203
C00766=1236.025,226.313,-58.208,-177.042,6.051,148.203
C00767=1236.029,226.064,-58.182,-177.045,6.049,148.203
C00768=1236.033,225.816,-58.158,-177.047,6.047,148.204
C00769=1236.037,225.567,-58.133,-177.050,6.045,148.204
C00770=1236.042,225.319,-58.107,-177.052,6.044,148.204
C00771=1236.047,225.069,-58.082,-177.054,6.042,148.205
C00772=1236.052,224.821,-58.057,-177.057,6.040,148.205
C00773=1236.055,224.572,-58.032,-177.060,6.039,148.205
C00774=1236.060,224.324,-58.007,-177.062,6.037,148.206
C00775=1236.065,224.075,-57.982,-177.065,6.035,148.206
C00776=1236.070,223.827,-57.957,-177.067,6.034,148.206
C00777=1236.073,223.578,-57.932,-177.070,6.032,148.207
C00778=1236.078,223.329,-57.907,-177.072,6.030,148.207
C00779=1236.083,223.080,-57.882,-177.075,6.028,148.207
C00780=1236.088,222.831,-57.857,-177.078,6.026,148.208
C00781=1236.091,222.583,-57.832,-177.080,6.025,148.208
C00782=1236.096,222.334,-57.807,-177.082,6.023,148.208
C00783=1236.101,222.085,-57.782,-177.085,6.022,148.209
C00784=1236.106,221.837,-57.757,-177.087,6.020,148.209
C00785=1236.110,221.587,-57.732,-177.090,6.018,148.209
C00786=1236.114,221.339,-57.707,-177.092,6.017,148.210
C00787=1236.120,221.091,-57.682,-177.095,6.015,148.210
C00788=1236.123,220.841,-57.658,-177.097,6.013,148.210
C00789=1236.128,220.593,-57.632,-177.100,6.011,148.211
C00790=1236.133,220.344,-57.607,-177.103,6.010,148.211
C00791=1236.137,220.096,-57.583,-177.105,6.008,148.211
C00792=1236.142,219.846,-57.558,-177.108,6.007,148.212
C00793=1236.146,219.598,-57.533,-177.110,6.005,148.212
C00794=1236.151,219.350,-57.509,-177.113,6.003,148.212
C00795=1236.155,219.100,-57.484,-177.116,6.001,148.213
C00796=1236.160,218.852,-57.460,-177.118,6.000,148.213
C00797=1236.164,218.603,-57.434,-177.120,5.998,148.213
C00798=1236.169,218.354,-57.409,-177.123,5.996,148.214
C00799=1236.174,218.106,-57.385,-177.126,5.994,148.214
C00800=1236.178,217.856,-57.360,-177.128,5.993,148.214
C00801=1236.182,217.609,-57.335,-177.130,5.991,148.215
C00802=1236.187,217.360,-57.311,-177.133,5.990,148.215
C00803=1236.192,217.110,-57.286,-177.136,5.988,148.216
C00804=1236.196,216.862,-57.262,-177.139,5.986,148.216
C00805=1236.201,216.613,-57.237,-177.141,5.985,148.216
C00806=1236.205,216.364,-57.213,-177.143,5.983,148.217
C00807=1236.210,216.115,-57.188,-177.146,5.981,148.217
C00808=1236.214,215.867,-57.163,-177.149,5.979,148.217
C00809=1236.219,215.618,-57.138,-177.151,5.978,148.218
C00810=1236.223,215.370,-57.114,-177.153,5.977,148.218
C00811=1236.228,215.120,-57.089,-177.156,5.975,148.218
C00812=1236.232,214.872,-57.065,-177.159,5.973,148.219
C00813=1236.237,214.623,-57.040,-177.161,5.971,148.219
C00814=1236.241,214.374,-57.016,-177.164,5.970,148.220
C00815=1236.246,214.125,-56.991,-177.166,5.968,148.220
C00816=1236.251,213.877,-56.967,-177.169,5.966,148.220
C00817=1236.256,213.628,-56.942,-177.172,5.965,148.221
C00818=1236.260,213.379,-56.918,-177.174,5.964,148.221
C00819=1236.265,213.130,-56.893,-177.176,5.962,148.221
C00820=1236.269,212.882,-56.869,-177.179,5.960,148.222
C00821=1236.274,212.633,-56.844,-177.182,5.958,148.222
C00822=1236.278,212.384,-56.820,-177.184,5.957,148.222
C00823=1236.283,212.114,-56.793,-177.187,5.955,148.223
C00824=1236.288,211.844,-56.767,-177.189,5.954,148.223
C00825=1236.292,211.573,-56.741,-177.192,5.952,148.224
C00826=1236.298,211.303,-56.714,-177.195,5.950,148.224
C00827=1236.303,211.054,-56.689,-177.198,5.948,148.224
C00828=1236.307,210.805,-56.665,-177.200,5.946,148.225
C00829=1236.311,210.556,-56.641,-177.203,5.944,148.225
C00830=1236.316,210.308,-56.616,-177.205,5.943,148.226
C00831=1236.320,210.059,-56.592,-177.208,5.942,148.226
C00832=1236.325,209.811,-56.568,-177.210,5.940,148.226
C00833=1236.330,209.561,-56.544,-177.213,5.938,148.227
C00834=1236.334,209.312,-56.520,-177.216,5.937,148.227
C00835=1236.339,209.064,-56.495,-177.218,5.935,148.227
C00836=1236.344,208.815,-56.471,-177.221,5.933,148.228
C00837=1236.347,208.566,-56.447,-177.223,5.932,148.228
C00838=1236.353,208.317,-56.422,-177.225,5.931,148.228
C00839=1236.357,208.068,-56.399,-177.228,5.929,148.229
C00840=1236.362,207.820,-56.374,-177.231,5.927,148.229
C00841=1236.366,207.571,-56.350,-177.233,5.926,148.230
C00842=1236.371,207.322,-56.325,-177.236,5.924,148.230
C00843=1236.375,207.073,-56.302,-177.239,5.922,148.230
C00844=1236.380,206.825,-56.278,-177.241,5.920,148.231
C00845=1236.385,206.576,-56.253,-177.243,5.919,148.231
C00846=1236.389,206.327,-56.229,-177.246,5.918,148.231
C00847=1236.394,206.078,-56.206,-177.249,5.916,148.232
C00848=1236.398,205.829,-56.181,-177.251,5.915,148.232
C00849=1236.403,205.581,-56.157,-177.254,5.913,148.233
C00850=1236.407,205.332,-56.133,-177.256,5.911,148.233
C00851=1236.412,205.083,-56.109,-177.259,5.909,148.233
C00852=1236.416,204.835,-56.085,-177.261,5.908,148.234
C00853=1236.421,204.586,-56.062,-177.264,5.906,148.234
C00854=1236.425,204.336,-56.037,-177.267,5.905,148.235
C00855=1236.430,204.088,-56.013,-177.269,5.904,148.235
C00856=1236.435,203.839,-55.989,-177.272,5.902,148.235
C00857=1236.439,203.590,-55.965,-177.274,5.900,148.236
C00858=1236.444,203.341,-55.942,-177.276,5.899,148.236
C00859=1236.449,203.093,-55.917,-177.279,5.897,148.236
C00860=1236.453,202.844,-55.893,-177.282,5.896,148.237
C00861=1236.457,202.595,-55.869,-177.285,5.894,148.237
C00862=1236.462,202.346,-55.845,-177.287,5.893,148.238
C00863=1236.466,202.097,-55.822,-177.289,5.891,148.238
C00864=1236.471,201.849,-55.798,-177.292,5.889,148.238
C00865=1236.476,201.599,-55.774,-177.294,5.888,148.239
C00866=1236.481,201.351,-55.750,-177.297,5.887,148.239
C00867=1236.485,201.102,-55.727,-177.300,5.885,148.240
C00868=1236.490,200.853,-55.702,-177.302,5.884,148.240
C00869=1236.494,200.604,-55.679,-177.304,5.882,148.240
C00870=1236.499,200.356,-55.655,-177.307,5.880,148.241
C00871=1236.504,200.107,-55.632,-177.310,5.879,148.241
C00872=1236.507,199.858,-55.607,-177.312,5.877,148.242
C00873=1236.512,199.609,-55.584,-177.315,5.876,148.242
C00874=1236.516,199.360,-55.560,-177.317,5.874,148.242
C00875=1236.522,199.111,-55.536,-177.320,5.873,148.243
C00876=1236.527,198.862,-55.512,-177.323,5.871,148.243
C00877=1236.531,198.614,-55.488,-177.325,5.870,148.244
C00878=1236.536,198.365,-55.465,-177.328,5.868,148.244
C00879=1236.540,198.116,-55.441,-177.330,5.866,148.244
C00880=1236.545,197.867,-55.418,-177.332,5.865,148.245
C00881=1236.549,197.618,-55.394,-177.335,5.864,148.245
C00882=1236.554,197.370,-55.370,-177.338,5.862,148.246
C00883=1236.559,197.121,-55.347,-177.340,5.861,148.246
C00884=1236.563,196.872,-55.323,-177.343,5.859,148.246
C00885=1236.568,196.623,-55.299,-177.345,5.857,148.247
C00886=1236.572,196.374,-55.276,-177.348,5.856,148.247
C00887=1236.577,196.125,-55.253,-177.351,5.855,148.248
C00888=1236.581,195.877,-55.229,-177.353,5.853,148.248
C00889=1236.586,195.628,-55.205,-177.355,5.852,148.248
C00890=1236.591,195.379,-55.182,-177.358,5.850,148.249
C00891=1236.596,195.130,-55.159,-177.360,5.849,148.249
C00892=1236.600,194.881,-55.134,-177.363,5.847,148.250
C00893=1236.605,194.632,-55.111,-177.366,5.845,148.250
C00894=1236.609,194.383,-55.088,-177.368,5.844,148.250
C00895=1236.613,194.134,-55.065,-177.370,5.843,148.251
C00896=1236.618,193.886,-55.041,-177.374,5.841,148.251
C00897=1236.622,193.637,-55.018,-177.376,5.840,148.252
C00898=1236.627,193.388,-54.994,-177.378,5.838,148.252
C00899=1236.632,193.139,-54.971,-177.381,5.836,148.252
C00900=1236.636,192.890,-54.947,-177.384,5.836,148.253
C00901=1236.641,192.641,-54.924,-177.386,5.834,148.253
C00902=1236.646,192.392,-54.900,-177.388,5.833,148.254
C00903=1236.650,192.143,-54.877,-177.391,5.831,148.254
C00904=1236.654,191.895,-54.854,-177.394,5.829,148.255
C00905=1236.660,191.646,-54.831,-177.396,5.828,148.255
C00906=1236.664,191.397,-54.808,-177.399,5.826,148.255
C00907=1236.669,191.148,-54.784,-177.401,5.825,148.256
C00908=1236.674,190.899,-54.761,-177.404,5.824,148.256
C00909=1236.678,190.650,-54.737,-177.407,5.822,148.257
C00910=1236.683,190.401,-54.714,-177.409,5.821,148.257
C00911=1236.687,190.152,-54.691,-177.411,5.819,148.257
C00912=1236.691,189.904,-54.667,-177.414,5.818,148.258
C00913=1236.696,189.655,-54.644,-177.417,5.817,148.258
C00914=1236.701,189.406,-54.621,-177.419,5.815,148.259
C00915=1236.705,189.157,-54.597,-177.421,5.814,148.259
C00916=1236.710,188.909,-54.575,-177.424,5.812,148.260
C00917=1236.715,188.660,-54.551,-177.427,5.810,148.260
C00918=1236.719,188.411,-54.528,-177.429,5.809,148.260
C00919=1236.724,188.162,-54.505,-177.432,5.807,148.261
C00920=1236.728,187.913,-54.482,-177.434,5.807,148.261
C00921=1236.733,187.663,-54.459,-177.437,5.805,148.262
C00922=1236.738,187.414,-54.436,-177.440,5.803,148.262
C00923=1236.743,187.166,-54.413,-177.442,5.802,148.262
C00924=1236.747,186.917,-54.390,-177.445,5.801,148.263
C00925=1236.752,186.668,-54.367,-177.447,5.800,148.263
C00926=1236.756,186.419,-54.343,-177.450,5.798,148.264
C00927=1236.762,186.150,-54.318,-177.453,5.796,148.264
C00928=1236.766,185.880,-54.294,-177.455,5.794,148.264
C00929=1236.772,185.610,-54.269,-177.458,5.794,148.265
C00930=1236.777,185.341,-54.243,-177.461,5.792,148.265
C00931=1236.781,185.092,-54.221,-177.463,5.790,148.266
C00932=1236.786,184.843,-54.198,-177.466,5.789,148.266
C00933=1236.790,184.594,-54.174,-177.468,5.787,148.267
C00934=1236.794,184.345,-54.152,-177.470,5.786,148.267
C00935=1236.800,184.097,-54.129,-177.473,5.784,148.267
C00936=1236.804,183.848,-54.105,-177.476,5.783,148.268
C00937=1236.809,183.598,-54.083,-177.478,5.782,148.268
C00938=1236.813,183.349,-54.060,-177.481,5.780,148.269
C00939=1236.817,183.101,-54.037,-177.484,5.779,148.269
C00940=1236.823,182.852,-54.014,-177.486,5.778,148.270
C00941=1236.828,182.603,-53.992,-177.488,5.776,148.270
C00942=1236.832,182.354,-53.969,-177.491,5.775,148.270
C00943=1236.836,182.105,-53.945,-177.494,5.773,148.271
C00944=1236.842,181.857,-53.922,-177.496,5.772,148.271
C00945=1236.846,181.607,-53.900,-177.499,5.770,148.272
C00946=1236.850,181.358,-53.877,-177.501,5.770,148.272
C00947=1236.854,181.109,-53.854,-177.504,5.768,148.273
C00948=1236.860,180.861,-53.832,-177.506,5.767,148.273
C00949=1236.864,180.612,-53.809,-177.509,5.765,148.273
C00950=1236.869,180.363,-53.786,-177.511,5.764,148.274
C00951=1236.874,180.113,-53.763,-177.514,5.762,148.274
C00952=1236.878,179.865,-53.741,-177.516,5.761,148.275
C00953=1236.883,179.616,-53.717,-177.519,5.760,148.275
C00954=1236.887,179.367,-53.695,-177.522,5.758,148.276
C00955=1236.892,179.118,-53.672,-177.524,5.757,148.276
C00956=1236.897,178.869,-53.650,-177.527,5.755,148.277
C00957=1236.902,178.620,-53.627,-177.529,5.754,148.277
C00958=1236.905,178.371,-53.604,-177.532,5.753,148.277
C00959=1236.911,178.122,-53.582,-177.534,5.752,148.278
C00960=1236.915,177.874,-53.559,-177.537,5.750,148.278
C00961=1236.920,177.624,-53.537,-177.539,5.749,148.279
C00962=1236.925,177.376,-53.514,-177.542,5.747,148.279
C00963=1236.930,177.126,-53.492,-177.544,5.746,148.280
C00964=1236.934,176.878,-53.469,-177.547,5.745,148.280
C00965=1236.938,176.628,-53.447,-177.550,5.744,148.281
C00966=1236.943,176.380,-53.424,-177.552,5.742,148.281
C00967=1236.947,176.131,-53.402,-177.554,5.741,148.281
C00968=1236.952,175.882,-53.378,-177.557,5.739,148.282
C00969=1236.957,175.633,-53.357,-177.560,5.739,148.282
C00970=1236.962,175.384,-53.333,-177.562,5.737,148.283
C00971=1236.966,175.135,-53.311,-177.565,5.735,148.283
C00972=1236.971,174.887,-53.289,-177.567,5.734,148.284
C00973=1236.976,174.637,-53.266,-177.570,5.732,148.284
C00974=1236.980,174.389,-53.244,-177.573,5.732,148.285
C00975=1236.985,174.139,-53.221,-177.575,5.730,148.285
C00976=1236.989,173.890,-53.198,-177.577,5.729,148.285
C00977=1236.994,173.642,-53.177,-177.580,5.727,148.286
C00978=1236.999,173.392,-53.154,-177.583,5.726,148.286
C00979=1237.003,173.143,-53.131,-177.585,5.724,148.287
C00980=1237.008,172.895,-53.110,-177.588,5.724,148.287
C00981=1237.013,172.645,-53.087,-177.590,5.722,148.288
C00982=1237.017,172.397,-53.065,-177.593,5.721,148.288
C00983=1237.022,172.148,-53.043,-177.596,5.719,148.289
C00984=1237.027,171.898,-53.020,-177.598,5.718,148.289
C00985=1237.031,171.650,-52.997,-177.600,5.716,148.289
C00986=1237.035,171.401,-52.975,-177.603,5.716,148.290
C00987=1237.041,171.152,-52.953,-177.606,5.714,148.290
C00988=1237.045,170.903,-52.930,-177.608,5.713,148.291
C00989=1237.049,170.654,-52.908,-177.611,5.711,148.291
C00990=1237.055,170.405,-52.886,-177.613,5.710,148.292
C00991=1237.059,170.155,-52.864,-177.616,5.710,148.292
C00992=1237.064,169.907,-52.842,-177.618,5.708,148.293
C00993=1237.068,169.658,-52.820,-177.620,5.707,148.293
C00994=1237.074,169.409,-52.797,-177.623,5.705,148.294
C00995=1237.078,169.160,-52.775,-177.626,5.704,148.294
C00996=1237.082,168.911,-52.752,-177.628,5.703,148.295
C00997=1237.087,168.662,-52.731,-177.631,5.702,148.295
C00998=1237.092,168.413,-52.708,-177.633,5.700,148.295
C00999=1237.097,168.164,-52.686,-177.636,5.699,148.296
C01000=1237.101,167.915,-52.664,-177.639,5.697,148.296
C01001=1237.105,167.667,-52.642,-177.641,5.696,148.297
C01002=1237.110,167.417,-52.619,-177.644,5.695,148.297
C01003=1237.115,167.169,-52.598,-177.646,5.694,148.298
C01004=1237.120,166.919,-52.576,-177.649,5.692,148.298
C01005=1237.124,166.671,-52.554,-177.651,5.691,148.299
C01006=1237.129,166.421,-52.532,-177.654,5.690,148.299
C01007=1237.134,166.172,-52.510,-177.656,5.689,148.300
C01008=1237.139,165.923,-52.488,-177.659,5.688,148.300
C01009=1237.143,165.674,-52.466,-177.661,5.686,148.301
C01010=1237.147,165.426,-52.443,-177.664,5.685,148.301
C01011=1237.152,165.177,-52.421,-177.666,5.684,148.302
C01012=1237.157,164.928,-52.399,-177.669,5.683,148.302
C01013=1237.161,164.679,-52.378,-177.672,5.681,148.302
C01014=1237.166,164.429,-52.355,-177.674,5.680,148.303
C01015=1237.171,164.181,-52.333,-177.677,5.679,148.303
C01016=1237.176,163.931,-52.311,-177.679,5.677,148.304
C01017=1237.180,163.683,-52.290,-177.682,5.676,148.304
C01018=1237.185,163.433,-52.268,-177.684,5.675,148.305
C01019=1237.190,163.185,-52.246,-177.686,5.674,148.305
C01020=1237.194,162.936,-52.224,-177.690,5.672,148.306
C01021=1237.199,162.687,-52.202,-177.692,5.671,148.306
C01022=1237.204,162.438,-52.181,-177.695,5.670,148.307
C01023=1237.209,162.188,-52.158,-177.697,5.669,148.307
C01024=1237.213,161.940,-52.136,-177.700,5.667,148.308
C01025=1237.218,161.690,-52.114,-177.702,5.666,148.308
C01026=1237.223,161.441,-52.093,-177.704,5.665,148.309
C01027=1237.228,161.192,-52.071,-177.707,5.664,148.309
C01028=1237.232,160.943,-52.049,-177.709,5.663,148.310
C01029=1237.237,160.695,-52.028,-177.712,5.661,148.310
C01030=1237.241,160.445,-52.006,-177.715,5.660,148.311
C01031=1237.247,160.176,-51.982,-177.717,5.659,148.311
C01032=1237.251,159.907,-51.959,-177.720,5.658,148.312
C01033=1237.257,159.638,-51.936,-177.723,5.656,148.312
C01034=1237.262,159.369,-51.911,-177.726,5.655,148.312
C01035=1237.266,159.119,-51.890,-177.728,5.654,148.313
C01036=1237.270,158.871,-51.869,-177.730,5.653,148.313
C01037=1237.275,158.622,-51.847,-177.734,5.651,148.314
C01038=1237.280,158.373,-51.825,-177.736,5.650,148.314
C01039=1237.284,158.124,-51.804,-177.738,5.649,148.315
C01040=1237.290,157.875,-51.783,-177.741,5.648,148.315
C01041=1237.294,157.626,-51.761,-177.743,5.647,148.316
C01042=1237.299,157.377,-51.739,-177.746,5.645,148.316
C01043=1237.303,157.128,-51.717,-177.748,5.644,148.317
C01044=1237.308,156.879,-51.696,-177.751,5.643,148.317
C01045=1237.313,156.630,-51.674,-177.754,5.642,148.318
C01046=1237.317,156.381,-51.652,-177.757,5.640,148.318
C01047=1237.322,156.132,-51.630,-177.759,5.639,148.319
C01048=1237.327,155.883,-51.610,-177.761,5.638,148.319
C01049=1237.332,155.633,-51.587,-177.764,5.637,148.320
C01050=1237.337,155.385,-51.566,-177.766,5.636,148.320
C01051=1237.341,155.136,-51.545,-177.769,5.635,148.321
C01052=1237.345,154.886,-51.523,-177.771,5.633,148.321
C01053=1237.350,154.638,-51.502,-177.774,5.633,148.322
C01054=1237.355,154.388,-51.481,-177.777,5.631,148.322
C01055=1237.360,154.140,-51.459,-177.779,5.630,148.323
C01056=1237.364,153.890,-51.437,-177.781,5.629,148.323
C01057=1237.370,153.641,-51.416,-177.784,5.628,148.324
C01058=1237.374,153.393,-51.395,-177.787,5.627,148.324
C01059=1237.378,153.144,-51.373,-177.789,5.625,148.325
C01060=1237.383,152.894,-51.352,-177.792,5.624,148.325
C01061=1237.388,152.646,-51.330,-177.794,5.623,148.326
C01062=1237.393,152.396,-51.309,-177.797,5.622,148.326
C01063=1237.397,152.147,-51.287,-177.799,5.621,148.327
C01064=1237.402,151.898,-51.267,-177.802,5.620,148.327
C01065=1237.407,151.649,-51.245,-177.804,5.618,148.328
C01066=1237.411,151.400,-51.223,-177.807,5.618,148.328
C01067=1237.416,151.151,-51.202,-177.810,5.616,148.329
C01068=1237.421,150.902,-51.180,-177.812,5.615,148.329
C01069=1237.426,150.653,-51.160,-177.814,5.614,148.330
C01070=1237.430,150.404,-51.138,-177.817,5.613,148.330
C01071=1237.435,150.155,-51.117,-177.820,5.612,148.331
C01072=1237.440,149.906,-51.095,-177.822,5.611,148.331
C01073=1237.444,149.657,-51.075,-177.825,5.609,148.332
C01074=1237.449,149.407,-51.054,-177.827,5.608,148.332
C01075=1237.454,149.158,-51.032,-177.830,5.607,148.333
C01076=1237.459,148.909,-51.011,-177.833,5.606,148.333
C01077=1237.463,148.661,-50.990,-177.835,5.605,148.334
C01078=1237.468,148.412,-50.969,-177.837,5.603,148.334
C01079=1237.472,148.162,-50.947,-177.840,5.602,148.335
C01080=1237.477,147.913,-50.927,-177.842,5.601,148.335
C01081=1237.482,147.664,-50.906,-177.845,5.600,148.336
C01082=1237.487,147.415,-50.884,-177.847,5.599,148.336
C01083=1237.491,147.167,-50.864,-177.850,5.598,148.337
C01084=1237.496,146.917,-50.842,-177.853,5.596,148.337
C01085=1237.501,146.668,-50.821,-177.855,5.596,148.338
C01086=1237.505,146.419,-50.800,-177.857,5.595,148.338
C01087=1237.510,146.170,-50.778,-177.861,5.593,148.339
C01088=1237.515,145.921,-50.758,-177.863,5.592,148.339
C01089=1237.520,145.672,-50.737,-177.865,5.592,148.340
C01090=1237.524,145.423,-50.715,-177.868,5.590,148.340
C01091=1237.529,145.173,-50.694,-177.870,5.589,148.341
C01092=1237.534,144.925,-50.674,-177.873,5.588,148.341
C01093=1237.539,144.675,-50.653,-177.876,5.587,148.342
C01094=1237.543,144.427,-50.632,-177.878,5.586,148.342
C01095=1237.548,144.178,-50.611,-177.880,5.585,148.343
C01096=1237.553,143.928,-50.589,-177.884,5.583,148.343
C01097=1237.557,143.679,-50.569,-177.886,5.583,148.344
C01098=1237.562,143.430,-50.547,-177.888,5.582,148.344
C01099=1237.566,143.181,-50.527,-177.891,5.580,148.345
C01100=1237.572,142.932,-50.506,-177.894,5.579,148.345
C01101=1237.577,142.683,-50.485,-177.896,5.578,148.346
C01102=1237.581,142.434,-50.464,-177.899,5.577,148.346
C01103=1237.586,142.185,-50.443,-177.901,5.576,148.347
C01104=1237.591,141.936,-50.423,-177.904,5.575,148.347
C01105=1237.595,141.686,-50.401,-177.906,5.574,148.348
C01106=1237.600,141.437,-50.381,-177.909,5.573,148.348
C01107=1237.605,141.188,-50.360,-177.911,5.572,148.349
C01108=1237.609,140.940,-50.339,-177.914,5.571,148.349
C01109=1237.614,140.690,-50.318,-177.916,5.569,148.350
C01110=1237.618,140.441,-50.298,-177.919,5.569,148.350
C01111=1237.624,140.192,-50.277,-177.921,5.568,148.351
C01112=1237.628,139.943,-50.256,-177.924,5.566,148.351
C01113=1237.633,139.694,-50.235,-177.926,5.565,148.352
C01114=1237.638,139.445,-50.215,-177.929,5.564,148.352
C01115=1237.643,139.196,-50.194,-177.932,5.563,148.353
C01116=1237.647,138.947,-50.174,-177.934,5.562,148.353
C01117=1237.652,138.697,-50.152,-177.937,5.561,148.354
C01118=1237.656,138.448,-50.132,-177.939,5.560,148.354
C01119=1237.661,138.199,-50.111,-177.942,5.559,148.355
C01120=1237.666,137.950,-50.090,-177.944,5.558,148.355
C01121=1237.671,137.701,-50.069,-177.947,5.557,148.356
C01122=1237.675,137.452,-50.048,-177.949,5.555,148.356
C01123=1237.680,137.203,-50.028,-177.952,5.555,148.357
C01124=1237.685,136.954,-50.007,-177.954,5.554,148.358
C01125=1237.689,136.705,-49.987,-177.957,5.553,148.358
C01126=1237.695,136.455,-49.966,-177.960,5.552,148.359
C01127=1237.699,136.206,-49.946,-177.962,5.551,148.359
C01128=1237.704,135.957,-49.926,-177.964,5.550,148.360
C01129=1237.709,135.708,-49.905,-177.967,5.548,148.360
C01130=1237.713,135.459,-49.884,-177.970,5.548,148.361
C01131=1237.718,135.210,-49.863,-177.972,5.547,148.361
C01132=1237.723,134.961,-49.843,-177.974,5.546,148.362
C01133=1237.727,134.712,-49.823,-177.977,5.544,148.362
C01134=1237.732,134.463,-49.802,-177.980,5.543,148.363
C01135=1237.737,134.195,-49.780,-177.982,5.543,148.363
C01136=1237.743,133.926,-49.758,-177.985,5.541,148.364
C01137=1237.747,133.657,-49.735,-177.988,5.540,148.364
C01138=1237.753,133.388,-49.714,-177.991,5.539,148.365
C01139=1237.758,133.139,-49.693,-177.993,5.538,148.366
C01140=1237.762,132.890,-49.673,-177.995,5.537,148.366
C01141=1237.767,132.640,-49.652,-177.999,5.536,148.367
C01142=1237.772,132.391,-49.632,-178.001,5.535,148.367
C01143=1237.776,132.142,-49.611,-178.003,5.534,148.368
C01144=1237.782,131.893,-49.591,-178.006,5.533,148.368
C01145=1237.786,131.644,-49.571,-178.009,5.532,148.369
C01146=1237.790,131.395,-49.550,-178.011,5.531,148.369
C01147=1237.795,131.146,-49.530,-178.013,5.530,148.370
C01148=1237.800,130.897,-49.509,-178.016,5.529,148.370
C01149=1237.805,130.648,-49.490,-178.019,5.528,148.371
C01150=1237.810,130.399,-49.469,-178.021,5.527,148.371
C01151=1237.814,130.150,-49.449,-178.024,5.526,148.372
C01152=1237.819,129.900,-49.428,-178.026,5.525,148.373
C01153=1237.824,129.651,-49.408,-178.029,5.524,148.373
C01154=1237.829,129.402,-49.388,-178.031,5.523,148.374
C01155=1237.833,129.153,-49.368,-178.034,5.522,148.374
C01156=1237.838,128.903,-49.347,-178.036,5.521,148.375
C01157=1237.843,128.654,-49.327,-178.038,5.520,148.375
C01158=1237.847,128.405,-49.307,-178.042,5.519,148.376
C01159=1237.852,128.156,-49.287,-178.044,5.518,148.376
C01160=1237.857,127.907,-49.267,-178.046,5.517,148.377
C01161=1237.862,127.658,-49.246,-178.049,5.517,148.378
C01162=1237.867,127.409,-49.226,-178.052,5.515,148.378
C01163=1237.871,127.160,-49.206,-178.054,5.514,148.379
C01164=1237.876,126.911,-49.186,-178.056,5.513,148.379
C01165=1237.881,126.661,-49.166,-178.059,5.513,148.380
C01166=1237.885,126.412,-49.146,-178.062,5.511,148.380
C01167=1237.891,126.163,-49.126,-178.064,5.510,148.381
C01168=1237.896,125.914,-49.105,-178.067,5.509,148.381
C01169=1237.900,125.665,-49.085,-178.069,5.509,148.382
C01170=1237.905,125.416,-49.065,-178.072,5.508,148.382
C01171=1237.909,125.167,-49.045,-178.075,5.506,148.383
C01172=1237.914,124.917,-49.025,-178.077,5.505,148.383
C01173=1237.918,124.668,-49.005,-178.079,5.505,148.384
C01174=1237.924,124.419,-48.986,-178.082,5.504,148.385
C01175=1237.928,124.170,-48.965,-178.085,5.502,148.385
C01176=1237.934,123.920,-48.945,-178.087,5.502,148.386
C01177=1237.938,123.671,-48.925,-178.089,5.501,148.386
C01178=1237.943,123.422,-48.905,-178.092,5.500,148.387
C01179=1237.948,123.174,-48.885,-178.095,5.499,148.387
C01180=1237.953,122.924,-48.865,-178.097,5.498,148.388
C01181=1237.957,122.675,-48.845,-178.100,5.497,148.388
C01182=1237.962,122.426,-48.825,-178.103,5.496,148.389
C01183=1237.966,122.177,-48.805,-178.105,5.495,148.389
C01184=1237.972,121.928,-48.786,-178.107,5.495,148.390
C01185=1237.976,121.679,-48.765,-178.110,5.493,148.390
C01186=1237.981,121.429,-48.746,-178.113,5.492,148.391
C01187=1237.986,121.180,-48.726,-178.115,5.492,148.392
C01188=1237.990,120.931,-48.705,-178.117,5.491,148.392
C01189=1237.995,120.682,-48.686,-178.120,5.490,148.393
C01190=1238.000,120.433,-48.666,-178.123,5.488,148.393
C01191=1238.004,120.183,-48.646,-178.125,5.488,148.394
C01192=1238.009,119.934,-48.627,-178.128,5.487,148.394
C01193=1238.014,119.685,-48.607,-178.130,5.486,148.395
C01194=1238.019,119.436,-48.587,-178.132,5.485,148.395
C01195=1238.024,119.186,-48.567,-178.136,5.484,148.396
C01196=1238.028,118.937,-48.547,-178.138,5.483,148.397
C01197=1238.034,118.689,-48.528,-178.140,5.482,148.397
C01198=1238.038,118.439,-48.508,-178.143,5.482,148.398
C01199=1238.043,118.190,-48.487,-178.145,5.481,148.398
C01200=1238.047,117.940,-48.468,-178.148,5.480,148.399
C01201=1238.053,117.692,-48.449,-178.151,5.478,148.399
C01202=1238.057,117.443,-48.428,-178.153,5.477,148.400
C01203=1238.062,117.193,-48.409,-178.156,5.477,148.400
C01204=1238.067,116.944,-48.389,-178.158,5.476,148.401
C01205=1238.071,116.695,-48.370,-178.160,5.475,148.402
C01206=1238.076,116.446,-48.350,-178.164,5.474,148.402
C01207=1238.081,116.197,-48.331,-178.166,5.473,148.403
C01208=1238.086,115.948,-48.311,-178.168,5.472,148.403
C01209=1238.091,115.698,-48.291,-178.171,5.471,148.404
C01210=1238.095,115.448,-48.272,-178.173,5.471,148.404
C01211=1238.100,115.200,-48.252,-178.176,5.470,148.405
C01212=1238.105,114.951,-48.232,-178.179,5.468,148.405
C01213=1238.110,114.701,-48.212,-178.181,5.468,148.406
C01214=1238.114,114.452,-48.194,-178.183,5.467,148.407
C01215=1238.119,114.203,-48.174,-178.186,5.466,148.407
C01216=1238.124,113.953,-48.154,-178.189,5.466,148.408
C01217=1238.129,113.705,-48.134,-178.191,5.465,148.408
C01218=1238.134,113.456,-48.115,-178.193,5.464,148.409
C01219=1238.138,113.206,-48.095,-178.197,5.462,148.410
C01220=1238.143,112.957,-48.076,-178.199,5.461,148.410
C01221=1238.148,112.708,-48.057,-178.201,5.461,148.411
C01222=1238.153,112.459,-48.037,-178.204,5.460,148.411
C01223=1238.158,112.209,-48.018,-178.206,5.459,148.412
C01224=1238.163,111.960,-47.998,-178.209,5.459,148.412
C01225=1238.167,111.711,-47.979,-178.212,5.457,148.413
C01226=1238.172,111.462,-47.959,-178.214,5.456,148.414
C01227=1238.176,111.213,-47.939,-178.217,5.456,148.414
C01228=1238.182,110.964,-47.920,-178.219,5.455,148.415
C01229=1238.186,110.715,-47.901,-178.222,5.454,148.415
C01230=1238.191,110.466,-47.882,-178.224,5.453,148.416
C01231=1238.196,110.216,-47.862,-178.227,5.453,148.416
C01232=1238.201,109.967,-47.842,-178.230,5.451,148.417
C01233=1238.205,109.718,-47.824,-178.232,5.450,148.417
C01234=1238.210,109.468,-47.804,-178.234,5.450,148.418
C01235=1238.215,109.220,-47.785,-178.237,5.449,148.419
C01236=1238.220,108.970,-47.765,-178.239,5.448,148.419
C01237=1238.224,108.721,-47.746,-178.242,5.447,148.420
C01238=1238.229,108.472,-47.727,-178.244,5.447,148.420
C01239=1238.235,108.203,-47.706,-178.248,5.445,148.421
C01240=1238.240,107.935,-47.686,-178.250,5.445,148.422
C01241=1238.245,107.666,-47.664,-178.253,5.444,148.422
C01242=1238.250,107.397,-47.643,-178.255,5.443,148.423
C01243=1238.255,107.149,-47.625,-178.258,5.442,148.423
C01244=1238.259,106.899,-47.605,-178.261,5.441,148.424
C01245=1238.265,106.650,-47.586,-178.263,5.440,148.425
C01246=1238.269,106.401,-47.567,-178.265,5.439,148.425
C01247=1238.274,106.152,-47.548,-178.268,5.439,148.426
C01248=1238.279,105.902,-47.528,-178.271,5.438,148.426
C01249=1238.284,105.654,-47.510,-178.273,5.437,148.427
C01250=1238.288,105.404,-47.490,-178.275,5.436,148.427
C01251=1238.294,105.155,-47.471,-178.279,5.435,148.428
C01252=1238.298,104.905,-47.452,-178.281,5.434,148.429
C01253=1238.303,104.656,-47.433,-178.283,5.433,148.429
C01254=1238.308,104.407,-47.413,-178.286,5.433,148.430
C01255=1238.312,104.158,-47.394,-178.289,5.432,148.430
C01256=1238.318,103.909,-47.375,-178.291,5.431,148.431
C01257=1238.322,103.659,-47.357,-178.293,5.431,148.431
C01258=1238.327,103.410,-47.337,-178.296,5.430,148.432
C01259=1238.331,103.161,-47.318,-178.299,5.429,148.433
C01260=1238.337,102.912,-47.299,-178.301,5.428,148.433
C01261=1238.341,102.662,-47.279,-178.304,5.427,148.434
C01262=1238.346,102.413,-47.262,-178.306,5.426,148.434
C01263=1238.351,102.163,-47.242,-178.309,5.426,148.435
C01264=1238.356,101.915,-47.223,-178.311,5.425,148.435
C01265=1238.361,101.665,-47.205,-178.314,5.424,148.436
C01266=1238.365,101.416,-47.186,-178.316,5.423,148.437
C01267=1238.371,101.167,-47.166,-178.319,5.422,148.437
C01268=1238.375,100.918,-47.147,-178.321,5.422,148.438
C01269=1238.380,100.669,-47.129,-178.324,5.421,148.438
C01270=1238.384,100.419,-47.110,-178.326,5.421,148.439
C01271=1238.390,100.170,-47.090,-178.329,5.419,148.439
C01272=1238.394,99.921,-47.072,-178.332,5.418,148.440
C01273=1238.399,99.672,-47.053,-178.334,5.418,148.441
C01274=1238.403,99.422,-47.034,-178.337,5.417,148.441
C01275=1238.409,99.173,-47.015,-178.339,5.416,148.442
C01276=1238.413,98.924,-46.996,-178.342,5.415,148.443
C01277=1238.418,98.674,-46.977,-178.344,5.415,148.443
C01278=1238.423,98.426,-46.959,-178.347,5.414,148.444
C01279=1238.428,98.176,-46.939,-178.349,5.413,148.444
C01280=1238.433,97.927,-46.921,-178.352,5.412,148.445
C01281=1238.438,97.678,-46.902,-178.354,5.412,148.446
C01282=1238.442,97.428,-46.883,-178.357,5.411,148.446
C01283=1238.448,97.179,-46.864,-178.359,5.410,148.447
C01284=1238.452,96.929,-46.846,-178.362,5.409,148.447
C01285=1238.457,96.681,-46.827,-178.365,5.408,148.448
C01286=1238.462,96.431,-46.808,-178.367,5.408,148.449
C01287=1238.466,96.182,-46.789,-178.370,5.407,148.449
C01288=1238.472,95.933,-46.770,-178.372,5.406,148.450
C01289=1238.476,95.683,-46.752,-178.375,5.405,148.450
C01290=1238.481,95.435,-46.733,-178.377,5.405,148.451
C01291=1238.486,95.185,-46.714,-178.380,5.404,148.451
C01292=1238.491,94.935,-46.696,-178.382,5.403,148.452
C01293=1238.496,94.687,-46.677,-178.385,5.403,148.453
C01294=1238.501,94.437,-46.659,-178.387,5.402,148.453
C01295=1238.505,94.188,-46.640,-178.390,5.401,148.454
C01296=1238.510,93.939,-46.621,-178.392,5.400,148.454
C01297=1238.514,93.689,-46.602,-178.395,5.400,148.455
C01298=1238.519,93.440,-46.584,-178.397,5.399,148.456
C01299=1238.525,93.191,-46.565,-178.400,5.398,148.456
C01300=1238.529,92.942,-46.547,-178.402,5.398,148.457
C01301=1238.534,92.692,-46.529,-178.405,5.396,148.457
C01302=1238.539,92.443,-46.509,-178.408,5.395,148.458
C01303=1238.544,92.194,-46.491,-178.411,5.395,148.459
C01304=1238.548,91.945,-46.472,-178.413,5.394,148.459
C01305=1238.554,91.696,-46.454,-178.415,5.393,148.460
C01306=1238.558,91.446,-46.435,-178.418,5.393,148.460
C01307=1238.563,91.197,-46.417,-178.421,5.392,148.461
C01308=1238.568,90.948,-46.399,-178.423,5.391,148.462
C01309=1238.573,90.698,-46.380,-178.425,5.390,148.462
C01310=1238.577,90.449,-46.361,-178.428,5.390,148.463
C01311=1238.582,90.200,-46.343,-178.431,5.389,148.463
C01312=1238.588,89.951,-46.324,-178.433,5.389,148.464
C01313=1238.592,89.701,-46.305,-178.436,5.388,148.465
C01314=1238.597,89.452,-46.287,-178.438,5.387,148.465
C01315=1238.602,89.203,-46.269,-178.441,5.386,148.466
C01316=1238.607,88.954,-46.251,-178.443,5.386,148.466
C01317=1238.611,88.704,-46.232,-178.446,5.385,148.467
C01318=1238.616,88.455,-46.214,-178.448,5.385,148.468
C01319=1238.621,88.206,-46.196,-178.451,5.384,148.468
C01320=1238.626,87.957,-46.178,-178.453,5.383,148.469
C01321=1238.631,87.707,-46.158,-178.456,5.382,148.469
C01322=1238.636,87.458,-46.140,-178.458,5.382,148.470
C01323=1238.641,87.209,-46.122,-178.461,5.381,148.471
C01324=1238.645,86.959,-46.104,-178.463,5.380,148.471
C01325=1238.650,86.710,-46.086,-178.466,5.380,148.472
C01326=1238.655,86.461,-46.067,-178.468,5.379,148.473
C01327=1238.660,86.212,-46.049,-178.471,5.378,148.473
C01328=1238.665,85.962,-46.031,-178.473,5.377,148.474
C01329=1238.669,85.713,-46.012,-178.476,5.377,148.474
C01330=1238.674,85.463,-45.994,-178.478,5.376,148.475
C01331=1238.679,85.214,-45.976,-178.481,5.376,148.476
C01332=1238.684,84.966,-45.958,-178.484,5.375,148.476
C01333=1238.689,84.715,-45.939,-178.486,5.374,148.477
C01334=1238.694,84.466,-45.921,-178.488,5.373,148.477
C01335=1238.699,84.217,-45.903,-178.491,5.373,148.478
C01336=1238.704,83.968,-45.885,-178.494,5.372,148.479
C01337=1238.709,83.719,-45.867,-178.496,5.372,148.479
C01338=1238.713,83.469,-45.848,-178.499,5.371,148.480
C01339=1238.718,83.220,-45.830,-178.501,5.370,148.480
C01340=1238.723,82.971,-45.813,-178.504,5.369,148.481
C01341=1238.728,82.721,-45.795,-178.506,5.369,148.482
C01342=1238.733,82.472,-45.776,-178.509,5.368,148.482
C01343=1238.738,82.204,-45.757,-178.512,5.367,148.483
C01344=1238.743,81.935,-45.737,-178.515,5.366,148.484
C01345=1238.748,81.667,-45.718,-178.517,5.366,148.484
C01346=1238.754,81.399,-45.698,-178.520,5.365,148.485
C01347=1238.758,81.149,-45.680,-178.523,5.364,148.486
C01348=1238.763,80.900,-45.662,-178.525,5.364,148.486
C01349=1238.768,80.651,-45.644,-178.527,5.363,148.487
C01350=1238.773,80.401,-45.626,-178.530,5.362,148.487
C01351=1238.778,80.152,-45.608,-178.533,5.362,148.488
C01352=1238.782,79.903,-45.590,-178.535,5.361,148.489
C01353=1238.788,79.654,-45.571,-178.538,5.360,148.489
C01354=1238.792,79.404,-45.553,-178.540,5.360,148.490
C01355=1238.797,79.155,-45.535,-178.543,5.359,148.490
C01356=1238.802,78.905,-45.517,-178.545,5.358,148.491
C01357=1238.807,78.656,-45.499,-178.548,5.358,148.492
C01358=1238.811,78.407,-45.482,-178.550,5.357,148.492
C01359=1238.816,78.158,-45.464,-178.553,5.356,148.493
C01360=1238.821,77.908,-45.447,-178.556,5.356,148.494
C01361=1238.826,77.659,-45.429,-178.558,5.355,148.494
C01362=1238.831,77.409,-45.410,-178.560,5.354,148.495
C01363=1238.836,77.160,-45.392,-178.563,5.354,148.495
C01364=1238.840,76.911,-45.374,-178.566,5.353,148.496
C01365=1238.845,76.662,-45.356,-178.568,5.352,148.497
C01366=1238.850,76.413,-45.338,-178.571,5.352,148.497
C01367=1238.856,76.163,-45.321,-178.574,5.351,148.498
C01368=1238.860,75.914,-45.303,-178.576,5.350,148.498
C01369=1238.865,75.665,-45.285,-178.578,5.350,148.499
C01370=1238.870,75.415,-45.267,-178.581,5.349,148.500
C01371=1238.875,75.166,-45.249,-178.584,5.348,148.500
C01372=1238.880,74.917,-45.231,-178.586,5.349,148.501
C01373=1238.885,74.667,-45.214,-178.588,5.348,148.502
C01374=1238.889,74.418,-45.197,-178.591,5.347,148.502
C01375=1238.894,74.169,-45.179,-178.593,5.346,148.503
C01376=1238.899,73.919,-45.160,-178.596,5.346,148.504
C01377=1238.904,73.669,-45.143,-178.598,5.345,148.504
C01378=1238.909,73.420,-45.125,-178.601,5.345,148.505
C01379=1238.914,73.171,-45.107,-178.604,5.344,148.506
C01380=1238.919,72.922,-45.089,-178.606,5.343,148.506
C01381=1238.924,72.672,-45.072,-178.609,5.343,148.507
C01382=1238.928,72.423,-45.054,-178.611,5.342,148.507
C01383=1238.933,72.174,-45.036,-178.614,5.341,148.508
C01384=1238.938,71.924,-45.019,-178.616,5.341,148.509
C01385=1238.943,71.675,-45.001,-178.619,5.340,148.509
C01386=1238.948,71.426,-44.983,-178.621,5.339,148.510
C01387=1238.953,71.176,-44.966,-178.624,5.339,148.511
C01388=1238.957,70.927,-44.948,-178.627,5.338,148.511
C01389=1238.962,70.678,-44.931,-178.629,5.337,148.512
C01390=1238.968,70.428,-44.913,-178.631,5.337,148.512
C01391=1238.972,70.179,-44.895,-178.634,5.336,148.513
C01392=1238.977,69.930,-44.878,-178.636,5.336,148.514
C01393=1238.982,69.680,-44.861,-178.639,5.336,148.514
C01394=1238.987,69.431,-44.843,-178.641,5.335,148.515
C01395=1238.992,69.182,-44.825,-178.644,5.335,148.516
C01396=1238.997,68.932,-44.807,-178.647,5.334,148.516
C01397=1239.001,68.683,-44.790,-178.649,5.333,148.517
C01398=1239.006,68.434,-44.773,-178.651,5.332,148.517
C01399=1239.011,68.185,-44.755,-178.654,5.332,148.518
C01400=1239.016,67.935,-44.738,-178.657,5.331,148.519
C01401=1239.021,67.686,-44.720,-178.659,5.331,148.519
C01402=1239.026,67.437,-44.703,-178.662,5.330,148.520
C01403=1239.031,67.188,-44.685,-178.665,5.329,148.521
C01404=1239.036,66.938,-44.669,-178.667,5.329,148.521
C01405=1239.041,66.689,-44.651,-178.669,5.328,148.522
C01406=1239.046,66.439,-44.633,-178.672,5.327,148.522
C01407=1239.051,66.190,-44.615,-178.674,5.327,148.523
C01408=1239.055,65.940,-44.599,-178.677,5.327,148.524
C01409=1239.060,65.691,-44.581,-178.679,5.326,148.524
C01410=1239.065,65.441,-44.563,-178.682,5.326,148.525
C01411=1239.070,65.193,-44.546,-178.685,5.325,148.526
C01412=1239.075,64.943,-44.529,-178.687,5.325,148.526
C01413=1239.080,64.694,-44.511,-178.690,5.324,148.527
C01414=1239.084,64.444,-44.494,-178.692,5.323,148.528
C01415=1239.090,64.196,-44.477,-178.695,5.322,148.528
C01416=1239.095,63.946,-44.459,-178.697,5.322,148.529
C01417=1239.099,63.697,-44.442,-178.700,5.321,148.530
C01418=1239.104,63.447,-44.425,-178.703,5.321,148.530
C01419=1239.109,63.198,-44.408,-178.705,5.321,148.531
C01420=1239.114,62.949,-44.390,-178.707,5.320,148.532
C01421=1239.119,62.699,-44.373,-178.710,5.320,148.532
C01422=1239.123,62.449,-44.356,-178.712,5.319,148.533
C01423=1239.128,62.200,-44.338,-178.715,5.318,148.534
C01424=1239.134,61.951,-44.321,-178.717,5.318,148.534
C01425=1239.138,61.702,-44.304,-178.720,5.317,148.535
C01426=1239.144,61.452,-44.286,-178.723,5.316,148.535
C01427=1239.148,61.203,-44.270,-178.725,5.316,148.536
C01428=1239.153,60.954,-44.252,-178.728,5.315,148.537
C01429=1239.157,60.704,-44.235,-178.730,5.315,148.537
C01430=1239.163,60.454,-44.218,-178.732,5.315,148.538
C01431=1239.168,60.205,-44.201,-178.735,5.314,148.539
C01432=1239.173,59.956,-44.184,-178.738,5.314,148.539
C01433=1239.178,59.707,-44.166,-178.740,5.313,148.540
C01434=1239.182,59.457,-44.150,-178.743,5.312,148.540
C01435=1239.187,59.208,-44.132,-178.745,5.311,148.541
C01436=1239.192,58.959,-44.115,-178.748,5.311,148.542
C01437=1239.198,58.709,-44.098,-178.750,5.310,148.542
C01438=1239.202,58.460,-44.081,-178.753,5.310,148.543
C01439=1239.207,58.211,-44.063,-178.755,5.310,148.544
C01440=1239.211,57.961,-44.047,-178.758,5.309,148.544
C01441=1239.217,57.712,-44.030,-178.760,5.309,148.545
C01442=1239.222,57.463,-44.013,-178.763,5.308,148.546
C01443=1239.227,57.213,-43.996,-178.766,5.308,148.546
C01444=1239.231,56.964,-43.979,-178.768,5.307,148.547
C01445=1239.236,56.714,-43.961,-178.771,5.306,148.548
C01446=1239.241,56.465,-43.945,-178.773,5.305,148.548
C01447=1239.247,56.197,-43.926,-178.776,5.305,148.549
C01448=1239.251,55.928,-43.908,-178.779,5.305,148.550
C01449=1239.257,55.660,-43.890,-178.781,5.304,148.550
C01450=1239.262,55.391,-43.872,-178.784,5.303,148.551
C01451=1239.267,55.142,-43.855,-178.787,5.303,148.552
C01452=1239.272,54.893,-43.838,-178.789,5.303,148.552
C01453=1239.278,54.643,-43.821,-178.791,5.303,148.553
C01454=1239.282,54.394,-43.804,-178.794,5.302,148.554
C01455=1239.287,54.144,-43.786,-178.797,5.301,148.554
C01456=1239.292,53.896,-43.770,-178.799,5.301,148.555
C01457=1239.297,53.646,-43.753,-178.802,5.300,148.556
C01458=1239.302,53.396,-43.736,-178.804,5.299,148.556
C01459=1239.306,53.147,-43.719,-178.806,5.300,148.557
C01460=1239.312,52.898,-43.703,-178.809,5.299,148.558
C01461=1239.317,52.648,-43.686,-178.811,5.298,148.558
C01462=1239.321,52.399,-43.669,-178.814,5.298,148.559
C01463=1239.326,52.149,-43.652,-178.817,5.297,148.560
C01464=1239.331,51.900,-43.636,-178.819,5.297,148.560
C01465=1239.336,51.651,-43.619,-178.822,5.296,148.561
C01466=1239.341,51.401,-43.602,-178.825,5.295,148.562
C01467=1239.345,51.151,-43.585,-178.827,5.296,148.562
C01468=1239.351,50.903,-43.569,-178.829,5.295,148.563
C01469=1239.356,50.653,-43.551,-178.832,5.294,148.564
C01470=1239.360,50.403,-43.535,-178.835,5.294,148.564
C01471=1239.365,50.155,-43.518,-178.837,5.293,148.565
C01472=1239.371,49.905,-43.501,-178.840,5.293,148.566
C01473=1239.375,49.655,-43.485,-178.843,5.292,148.566
C01474=1239.380,49.406,-43.468,-178.845,5.292,148.567
C01475=1239.385,49.157,-43.451,-178.847,5.291,148.567
C01476=1239.390,48.907,-43.434,-178.849,5.291,148.568
C01477=1239.395,48.658,-43.418,-178.852,5.290,148.569
C01478=1239.400,48.409,-43.401,-178.855,5.290,148.569
C01479=1239.405,48.159,-43.384,-178.857,5.289,148.570
C01480=1239.410,47.910,-43.368,-178.859,5.289,148.571
C01481=1239.414,47.660,-43.352,-178.862,5.289,148.571
C01482=1239.420,47.410,-43.335,-178.865,5.288,148.572
C01483=1239.425,47.162,-43.318,-178.867,5.288,148.573
C01484=1239.429,46.912,-43.302,-178.870,5.287,148.573
C01485=1239.434,46.663,-43.285,-178.873,5.286,148.574
C01486=1239.440,46.414,-43.268,-178.875,5.287,148.575
C01487=1239.444,46.163,-43.252,-178.877,5.286,148.575
C01488=1239.449,45.914,-43.235,-178.880,5.286,148.576
C01489=1239.454,45.665,-43.219,-178.883,5.285,148.577
C01490=1239.459,45.415,-43.202,-178.885,5.284,148.577
C01491=1239.464,45.167,-43.186,-178.888,5.284,148.578
C01492=1239.469,44.917,-43.169,-178.890,5.284,148.579
C01493=1239.473,44.667,-43.153,-178.893,5.284,148.580
C01494=1239.479,44.418,-43.137,-178.895,5.283,148.580
C01495=1239.484,44.168,-43.119,-178.898,5.282,148.581
C01496=1239.489,43.920,-43.103,-178.900,5.282,148.582
C01497=1239.494,43.670,-43.087,-178.903,5.281,148.582
C01498=1239.498,43.420,-43.070,-178.905,5.281,148.583
C01499=1239.503,43.171,-43.054,-178.907,5.281,148.583
C01500=1239.508,42.922,-43.037,-178.910,5.280,148.584
C01501=1239.514,42.672,-43.021,-178.913,5.279,148.585
C01502=1239.518,42.423,-43.005,-178.915,5.279,148.585
C01503=1239.523,42.173,-42.988,-178.918,5.278,148.586
C01504=1239.528,41.924,-42.972,-178.920,5.278,148.587
C01505=1239.533,41.674,-42.956,-178.923,5.278,148.587
C01506=1239.538,41.425,-42.939,-178.925,5.277,148.588
C01507=1239.542,41.176,-42.923,-178.928,5.277,148.589
C01508=1239.548,40.926,-42.907,-178.930,5.276,148.589
C01509=1239.553,40.677,-42.890,-178.933,5.276,148.590
C01510=1239.557,40.427,-42.873,-178.935,5.276,148.591
C01511=1239.563,40.178,-42.858,-178.938,5.275,148.591
C01512=1239.567,39.928,-42.841,-178.940,5.275,148.592
C01513=1239.573,39.679,-42.825,-178.943,5.274,148.593
C01514=1239.577,39.430,-42.809,-178.946,5.274,148.593
C01515=1239.582,39.181,-42.792,-178.948,5.274,148.594
C01516=1239.587,38.931,-42.776,-178.950,5.273,148.595
C01517=1239.592,38.682,-42.760,-178.953,5.273,148.595
C01518=1239.597,38.431,-42.744,-178.956,5.272,148.596
C01519=1239.603,38.183,-42.727,-178.958,5.271,148.597
C01520=1239.607,37.933,-42.711,-178.960,5.272,148.598
C01521=1239.612,37.684,-42.695,-178.963,5.271,148.598
C01522=1239.617,37.434,-42.678,-178.966,5.271,148.599
C01523=1239.622,37.185,-42.663,-178.968,5.270,148.600
C01524=1239.627,36.935,-42.646,-178.971,5.269,148.600
C01525=1239.632,36.686,-42.630,-178.973,5.270,148.601
C01526=1239.637,36.437,-42.614,-178.976,5.269,148.602
C01527=1239.642,36.187,-42.598,-178.978,5.269,148.602
C01528=1239.646,35.938,-42.582,-178.981,5.268,148.603
C01529=1239.652,35.688,-42.566,-178.984,5.267,148.604
C01530=1239.656,35.439,-42.549,-178.986,5.268,148.604
C01531=1239.662,35.189,-42.534,-178.988,5.267,148.605
C01532=1239.666,34.940,-42.517,-178.991,5.267,148.606
C01533=1239.672,34.690,-42.501,-178.994,5.266,148.606
C01534=1239.676,34.441,-42.485,-178.996,5.265,148.607
C01535=1239.681,34.192,-42.469,-178.998,5.266,148.608
C01536=1239.686,33.942,-42.453,-179.001,5.265,148.608
C01537=1239.691,33.693,-42.437,-179.004,5.264,148.609
C01538=1239.696,33.444,-42.421,-179.006,5.264,148.610
C01539=1239.701,33.194,-42.405,-179.008,5.264,148.610
C01540=1239.706,32.945,-42.390,-179.011,5.264,148.611
C01541=1239.710,32.695,-42.373,-179.014,5.263,148.612
C01542=1239.716,32.446,-42.357,-179.016,5.262,148.612
C01543=1239.720,32.196,-42.341,-179.019,5.262,148.613
C01544=1239.726,31.947,-42.325,-179.021,5.262,148.614
C01545=1239.730,31.697,-42.309,-179.024,5.262,148.614
C01546=1239.735,31.448,-42.293,-179.026,5.261,148.615
C01547=1239.741,31.199,-42.277,-179.029,5.260,148.616
C01548=1239.746,30.949,-42.261,-179.031,5.261,148.616
C01549=1239.751,30.700,-42.245,-179.034,5.260,148.617
C01550=1239.755,30.450,-42.229,-179.036,5.260,148.618
C01551=1239.760,30.181,-42.213,-179.039,5.259,148.619
C01552=1239.766,29.913,-42.196,-179.042,5.258,148.619
C01553=1239.771,29.645,-42.179,-179.044,5.258,148.620
C01554=1239.776,29.375,-42.161,-179.047,5.258,148.621
C01555=1239.781,29.127,-42.145,-179.049,5.258,148.621
C01556=1239.787,28.877,-42.129,-179.052,5.257,148.622
C01557=1239.792,28.627,-42.113,-179.055,5.257,148.623
C01558=1239.797,28.378,-42.097,-179.057,5.256,148.623
C01559=1239.801,28.129,-42.082,-179.060,5.256,148.624
C01560=1239.806,27.879,-42.066,-179.062,5.256,148.625
C01561=1239.812,27.630,-42.051,-179.065,5.255,148.626
C01562=1239.817,27.380,-42.035,-179.067,5.255,148.626
C01563=1239.821,27.131,-42.018,-179.070,5.254,148.627
C01564=1239.827,26.881,-42.003,-179.072,5.255,148.628
C01565=1239.831,26.632,-41.987,-179.075,5.254,148.628
C01566=1239.836,26.382,-41.972,-179.077,5.253,148.629
C01567=1239.841,26.133,-41.955,-179.080,5.253,148.630
C01568=1239.846,25.883,-41.940,-179.082,5.253,148.630
C01569=1239.851,25.634,-41.925,-179.085,5.253,148.631
C01570=1239.856,25.385,-41.909,-179.087,5.252,148.632
C01571=1239.861,25.135,-41.893,-179.090,5.251,148.632
C01572=1239.866,24.885,-41.877,-179.092,5.252,148.633
C01573=1239.871,24.637,-41.862,-179.095,5.251,148.634
C01574=1239.875,24.387,-41.846,-179.097,5.251,148.634
C01575=1239.881,24.137,-41.830,-179.100,5.250,148.635
C01576=1239.886,23.888,-41.815,-179.102,5.250,148.636
C01577=1239.890,23.638,-41.799,-179.105,5.250,148.636
C01578=1239.896,23.389,-41.784,-179.107,5.249,148.637
C01579=1239.901,23.139,-41.768,-179.110,5.249,148.638
C01580=1239.906,22.890,-41.752,-179.112,5.249,148.638
C01581=1239.910,22.640,-41.737,-179.115,5.248,148.639
C01582=1239.916,22.391,-41.721,-179.117,5.248,148.640
C01583=1239.921,22.142,-41.705,-179.120,5.247,148.641
C01584=1239.925,21.892,-41.690,-179.122,5.247,148.641
C01585=1239.930,21.643,-41.674,-179.125,5.247,148.642
C01586=1239.936,21.393,-41.659,-179.127,5.246,148.643
C01587=1239.940,21.144,-41.644,-179.130,5.246,148.643
C01588=1239.945,20.894,-41.628,-179.132,5.246,148.644
C01589=1239.951,20.645,-41.612,-179.135,5.245,148.645
C01590=1239.955,20.396,-41.597,-179.137,5.245,148.645
C01591=1239.961,20.146,-41.582,-179.140,5.244,148.646
C01592=1239.965,19.896,-41.566,-179.142,5.245,148.647
C01593=1239.970,19.647,-41.551,-179.145,5.244,148.647
C01594=1239.975,19.398,-41.535,-179.147,5.243,148.648
C01595=1239.981,19.148,-41.519,-179.150,5.244,148.649
C01596=1239.985,18.898,-41.504,-179.152,5.243,148.649
C01597=1239.990,18.649,-41.488,-179.155,5.243,148.650
C01598=1239.996,18.400,-41.473,-179.158,5.242,148.651
C01599=1240.000,18.151,-41.458,-179.160,5.242,148.651
C01600=1240.005,17.900,-41.442,-179.163,5.242,148.652
C01601=1240.010,17.651,-41.427,-179.165,5.242,148.653
C01602=1240.015,17.402,-41.411,-179.168,5.241,148.654
C01603=1240.021,17.152,-41.396,-179.170,5.241,148.654
C01604=1240.025,16.903,-41.382,-179.173,5.241,148.655
C01605=1240.030,16.653,-41.366,-179.175,5.240,148.656
C01606=1240.035,16.404,-41.351,-179.177,5.240,148.656
C01607=1240.040,16.154,-41.335,-179.180,5.240,148.657
C01608=1240.045,15.905,-41.320,-179.183,5.239,148.658
C01609=1240.050,15.656,-41.304,-179.185,5.239,148.659
C01610=1240.055,15.406,-41.288,-179.187,5.239,148.659
C01611=1240.060,15.156,-41.274,-179.190,5.238,148.660
C01612=1240.065,14.907,-41.259,-179.193,5.238,148.661
C01613=1240.070,14.657,-41.244,-179.195,5.237,148.661
C01614=1240.075,14.408,-41.228,-179.198,5.238,148.662
C01615=1240.080,14.158,-41.213,-179.200,5.237,148.663
C01616=1240.085,13.909,-41.197,-179.203,5.237,148.663
C01617=1240.090,13.659,-41.183,-179.205,5.237,148.664
C01618=1240.095,13.410,-41.167,-179.208,5.236,148.665
C01619=1240.100,13.161,-41.152,-179.210,5.236,148.665
C01620=1240.105,12.911,-41.137,-179.213,5.235,148.666
C01621=1240.109,12.661,-41.121,-179.215,5.235,148.667
C01622=1240.115,12.411,-41.106,-179.218,5.235,148.667
C01623=1240.120,12.162,-41.091,-179.220,5.234,148.668
C01624=1240.125,11.913,-41.076,-179.222,5.235,148.669
C01625=1240.130,11.664,-41.061,-179.225,5.234,148.670
C01626=1240.135,11.414,-41.046,-179.228,5.234,148.670
C01627=1240.140,11.165,-41.031,-179.230,5.234,148.671
C01628=1240.145,10.915,-41.015,-179.233,5.234,148.672
C01629=1240.150,10.665,-41.001,-179.235,5.233,148.672
C01630=1240.154,10.416,-40.986,-179.238,5.232,148.673
C01631=1240.160,10.166,-40.970,-179.240,5.233,148.674
C01632=1240.164,9.917,-40.955,-179.243,5.232,148.675
C01633=1240.170,9.667,-40.940,-179.245,5.232,148.675
C01634=1240.175,9.418,-40.925,-179.248,5.232,148.676
C01635=1240.180,9.169,-40.910,-179.250,5.231,148.677
C01636=1240.185,8.919,-40.895,-179.253,5.231,148.677
C01637=1240.190,8.670,-40.880,-179.255,5.231,148.678
C01638=1240.195,8.420,-40.864,-179.258,5.231,148.679
C01639=1240.200,8.170,-40.850,-179.260,5.230,148.679
C01640=1240.205,7.921,-40.835,-179.263,5.229,148.680
C01641=1240.210,7.671,-40.820,-179.265,5.230,148.681
C01642=1240.215,7.422,-40.805,-179.268,5.229,148.681
C01643=1240.220,7.173,-40.790,-179.270,5.229,148.682
C01644=1240.225,6.923,-40.775,-179.273,5.229,148.683
C01645=1240.230,6.674,-40.760,-179.275,5.229,148.684
C01646=1240.235,6.424,-40.746,-179.278,5.228,148.684
C01647=1240.240,6.175,-40.731,-179.280,5.228,148.685
C01648=1240.245,5.926,-40.716,-179.283,5.228,148.686
C01649=1240.250,5.676,-40.701,-179.286,5.227,148.686
C01650=1240.255,5.426,-40.686,-179.288,5.228,148.687
C01651=1240.260,5.177,-40.671,-179.290,5.227,148.688
C01652=1240.265,4.927,-40.656,-179.293,5.227,148.688
C01653=1240.270,4.678,-40.642,-179.296,5.226,148.689
C01654=1240.274,4.428,-40.626,-179.298,5.226,148.690
C01655=1240.281,4.159,-40.610,-179.300,5.226,148.691
C01656=1240.286,3.891,-40.595,-179.303,5.226,148.691
C01657=1240.291,3.622,-40.579,-179.306,5.225,148.692
C01658=1240.297,3.353,-40.563,-179.308,5.225,148.693
C01659=1240.301,3.104,-40.548,-179.311,5.225,148.694
C01660=1240.306,2.854,-40.533,-179.313,5.224,148.694
C01661=1240.312,2.605,-40.518,-179.316,5.224,148.695
C01662=1240.317,2.355,-40.503,-179.319,5.224,148.696
C01663=1240.322,2.105,-40.489,-179.321,5.224,148.697
C01664=1240.326,1.856,-40.474,-179.323,5.224,148.697
C01665=1240.332,1.606,-40.459,-179.326,5.223,148.698
C01666=1240.337,1.357,-40.444,-179.329,5.223,148.699
C01667=1240.342,1.107,-40.430,-179.331,5.222,148.699
C01668=1240.346,0.858,-40.415,-179.333,5.223,148.700
C01669=1240.352,0.608,-40.400,-179.336,5.222,148.701
C01670=1240.357,0.358,-40.386,-179.339,5.222,148.701
C01671=1240.362,0.109,-40.371,-179.341,5.222,148.702
C01672=1240.367,-0.140,-40.357,-179.344,5.221,148.703
C01673=1240.371,-0.389,-40.342,-179.346,5.221,148.703
C01674=1240.377,-0.639,-40.327,-179.348,5.221,148.704
C01675=1240.382,-0.889,-40.312,-179.351,5.221,148.705
C01676=1240.386,-1.138,-40.297,-179.354,5.220,148.705
C01677=1240.391,-1.388,-40.283,-179.356,5.221,148.706
C01678=1240.396,-1.638,-40.269,-179.359,5.220,148.707
C01679=1240.402,-1.887,-40.253,-179.361,5.220,148.708
C01680=1240.407,-2.137,-40.239,-179.364,5.220,148.708
C01681=1240.412,-2.387,-40.225,-179.366,5.219,148.709
C01682=1240.416,-2.636,-40.210,-179.368,5.220,148.710
C01683=1240.421,-2.885,-40.196,-179.371,5.219,148.711
C01684=1240.426,-3.135,-40.181,-179.374,5.219,148.711
C01685=1240.432,-3.385,-40.166,-179.376,5.219,148.712
C01686=1240.437,-3.633,-40.152,-179.378,5.218,148.713
C01687=1240.442,-3.883,-40.137,-179.381,5.218,148.713
C01688=1240.447,-4.133,-40.123,-179.383,5.218,148.714
C01689=1240.452,-4.382,-40.108,-179.386,5.217,148.715
C01690=1240.457,-4.632,-40.094,-179.389,5.217,148.716
C01691=1240.462,-4.881,-40.080,-179.391,5.218,148.716
C01692=1240.467,-5.131,-40.065,-179.394,5.217,148.717
C01693=1240.472,-5.381,-40.051,-179.396,5.217,148.718
C01694=1240.477,-5.630,-40.035,-179.398,5.217,148.718
C01695=1240.482,-5.880,-40.021,-179.401,5.216,148.719
C01696=1240.487,-6.129,-40.007,-179.404,5.216,148.720
C01697=1240.492,-6.379,-39.993,-179.406,5.216,148.720
C01698=1240.497,-6.628,-39.979,-179.408,5.215,148.721
C01699=1240.502,-6.877,-39.964,-179.411,5.215,148.722
C01700=1240.507,-7.127,-39.949,-179.413,5.215,148.723
C01701=1240.512,-7.377,-39.935,-179.416,5.215,148.723
C01702=1240.517,-7.627,-39.921,-179.418,5.214,148.724
C01703=1240.522,-7.876,-39.907,-179.421,5.215,148.725
C01704=1240.527,-8.125,-39.893,-179.424,5.214,148.726
C01705=1240.532,-8.374,-39.878,-179.426,5.215,148.726
C01706=1240.537,-8.624,-39.863,-179.428,5.214,148.727
C01707=1240.542,-8.874,-39.849,-179.431,5.213,148.728
C01708=1240.547,-9.124,-39.835,-179.433,5.214,148.728
C01709=1240.552,-9.373,-39.821,-179.436,5.213,148.729
C01710=1240.557,-9.623,-39.806,-179.438,5.213,148.730
C01711=1240.562,-9.872,-39.792,-179.440,5.213,148.730
C01712=1240.567,-10.122,-39.778,-179.443,5.212,148.731
C01713=1240.572,-10.371,-39.764,-179.446,5.212,148.732
C01714=1240.577,-10.621,-39.750,-179.448,5.212,148.732
C01715=1240.582,-10.871,-39.735,-179.451,5.212,148.733
C01716=1240.588,-11.120,-39.721,-179.453,5.212,148.734
C01717=1240.592,-11.369,-39.706,-179.456,5.212,148.735
C01718=1240.597,-11.619,-39.692,-179.458,5.211,148.735
C01719=1240.602,-11.868,-39.678,-179.461,5.212,148.736
C01720=1240.607,-12.118,-39.664,-179.463,5.211,148.737
C01721=1240.612,-12.368,-39.649,-179.466,5.211,148.738
C01722=1240.618,-12.617,-39.635,-179.468,5.211,148.738
C01723=1240.623,-12.866,-39.621,-179.471,5.210,148.739
C01724=1240.628,-13.116,-39.607,-179.473,5.210,148.740
C01725=1240.633,-13.366,-39.593,-179.475,5.210,148.740
C01726=1240.638,-13.615,-39.579,-179.478,5.209,148.741
C01727=1240.643,-13.865,-39.564,-179.481,5.210,148.742
C01728=1240.648,-14.115,-39.551,-179.483,5.210,148.743
C01729=1240.653,-14.364,-39.537,-179.486,5.209,148.743
C01730=1240.658,-14.614,-39.523,-179.488,5.209,148.744
C01731=1240.663,-14.863,-39.509,-179.491,5.209,148.745
C01732=1240.668,-15.113,-39.495,-179.493,5.208,148.745
C01733=1240.673,-15.362,-39.480,-179.495,5.209,148.746
C01734=1240.678,-15.612,-39.466,-179.498,5.208,148.747
C01735=1240.684,-15.861,-39.452,-179.500,5.208,148.747
C01736=1240.689,-16.111,-39.438,-179.503,5.208,148.748
C01737=1240.693,-16.361,-39.424,-179.505,5.207,148.749
C01738=1240.698,-16.610,-39.410,-179.508,5.208,148.750
C01739=1240.703,-16.859,-39.396,-179.511,5.207,148.750
C01740=1240.709,-17.109,-39.383,-179.513,5.208,148.751
C01741=1240.713,-17.359,-39.368,-179.515,5.207,148.752
C01742=1240.719,-17.608,-39.354,-179.518,5.207,148.753
C01743=1240.724,-17.858,-39.340,-179.520,5.207,148.753
C01744=1240.728,-18.107,-39.326,-179.523,5.206,148.754
C01745=1240.733,-18.357,-39.312,-179.525,5.206,148.755
C01746=1240.739,-18.607,-39.299,-179.527,5.206,148.755
C01747=1240.744,-18.856,-39.285,-179.530,5.206,148.756
C01748=1240.749,-19.106,-39.270,-179.532,5.206,148.757
C01749=1240.754,-19.355,-39.257,-179.535,5.206,148.758
C01750=1240.759,-19.604,-39.243,-179.538,5.205,148.758
C01751=1240.764,-19.855,-39.229,-179.540,5.206,148.759
C01752=1240.769,-20.104,-39.215,-179.543,5.205,148.760
C01753=1240.774,-20.353,-39.201,-179.545,5.205,148.760
C01754=1240.779,-20.603,-39.187,-179.548,5.205,148.761
C01755=1240.784,-20.853,-39.173,-179.550,5.204,148.762
C01756=1240.789,-21.102,-39.160,-179.552,5.205,148.763
C01757=1240.794,-21.352,-39.146,-179.555,5.204,148.763
C01758=1240.799,-21.601,-39.132,-179.557,5.204,148.764
C01759=1240.805,-21.870,-39.117,-179.560,5.204,148.765
C01760=1240.810,-22.139,-39.102,-179.563,5.204,148.766
C01761=1240.816,-22.409,-39.087,-179.565,5.203,148.766
C01762=1240.821,-22.678,-39.072,-179.568,5.204,148.767
C01763=1240.827,-22.927,-39.058,-179.571,5.203,148.768
C01764=1240.831,-23.177,-39.045,-179.573,5.203,148.769
C01765=1240.836,-23.427,-39.031,-179.575,5.203,148.769
C01766=1240.842,-23.676,-39.017,-179.578,5.203,148.770
C01767=1240.847,-23.926,-39.004,-179.580,5.203,148.771
C01768=1240.851,-24.176,-38.990,-179.583,5.202,148.771
C01769=1240.857,-24.425,-38.976,-179.586,5.202,148.772
C01770=1240.862,-24.675,-38.962,-179.588,5.202,148.773
C01771=1240.867,-24.924,-38.949,-179.591,5.202,148.774
C01772=1240.872,-25.173,-38.935,-179.593,5.202,148.774
C01773=1240.877,-25.424,-38.921,-179.596,5.202,148.775
C01774=1240.882,-25.672,-38.908,-179.598,5.201,148.776
C01775=1240.887,-25.923,-38.894,-179.600,5.202,148.776
C01776=1240.892,-26.173,-38.880,-179.603,5.201,148.777
C01777=1240.897,-26.421,-38.867,-179.605,5.201,148.778
C01778=1240.902,-26.672,-38.853,-179.608,5.201,148.779
C01779=1240.908,-26.921,-38.839,-179.610,5.200,148.779
C01780=1240.912,-27.171,-38.826,-179.612,5.201,148.780
C01781=1240.917,-27.420,-38.812,-179.616,5.200,148.781
C01782=1240.922,-27.670,-38.800,-179.618,5.201,148.782
C01783=1240.927,-27.919,-38.785,-179.620,5.200,148.782
C01784=1240.933,-28.168,-38.771,-179.622,5.201,148.783
C01785=1240.937,-28.418,-38.758,-179.625,5.200,148.784
C01786=1240.943,-28.667,-38.744,-179.628,5.200,148.784
C01787=1240.948,-28.918,-38.731,-179.630,5.200,148.785
C01788=1240.952,-29.167,-38.717,-179.632,5.199,148.786
C01789=1240.958,-29.417,-38.704,-179.635,5.200,148.786
C01790=1240.962,-29.666,-38.690,-179.637,5.199,148.787
C01791=1240.968,-29.916,-38.677,-179.640,5.199,148.788
C01792=1240.972,-30.165,-38.663,-179.642,5.199,148.789
C01793=1240.978,-30.415,-38.650,-179.645,5.199,148.789
C01794=1240.983,-30.664,-38.636,-179.647,5.199,148.790
C01795=1240.988,-30.914,-38.623,-179.650,5.199,148.791
C01796=1240.993,-31.163,-38.609,-179.652,5.199,148.792
C01797=1240.998,-31.413,-38.597,-179.655,5.198,148.792
C01798=1241.004,-31.663,-38.583,-179.657,5.198,148.793
C01799=1241.008,-31.913,-38.569,-179.659,5.198,148.794
C01800=1241.014,-32.162,-38.556,-179.662,5.198,148.794
C01801=1241.018,-32.412,-38.542,-179.665,5.198,148.795
C01802=1241.024,-32.661,-38.529,-179.667,5.198,148.796
C01803=1241.028,-32.911,-38.516,-179.670,5.197,148.797
C01804=1241.034,-33.160,-38.502,-179.672,5.198,148.797
C01805=1241.038,-33.410,-38.489,-179.675,5.197,148.798
C01806=1241.044,-33.659,-38.475,-179.677,5.197,148.799
C01807=1241.049,-33.909,-38.462,-179.679,5.197,148.799
C01808=1241.054,-34.159,-38.449,-179.681,5.197,148.800
C01809=1241.059,-34.408,-38.436,-179.684,5.197,148.801
C01810=1241.064,-34.658,-38.422,-179.687,5.196,148.802
C01811=1241.069,-34.908,-38.409,-179.689,5.197,148.803
C01812=1241.075,-35.157,-38.396,-179.692,5.196,148.803
C01813=1241.079,-35.407,-38.383,-179.694,5.197,148.804
C01814=1241.085,-35.657,-38.369,-179.697,5.196,148.805
C01815=1241.089,-35.906,-38.356,-179.699,5.196,148.805
C01816=1241.095,-36.156,-38.343,-179.702,5.196,148.806
C01817=1241.100,-36.405,-38.330,-179.704,5.195,148.807
